LIN {X 0,Y 573.207,Z 217.084,A -85,B 0,C 180,E1 -2298.541,E2 -2298.541} C_VEL
LIN {X 0,Y 573.23,Z 217.078,A -85,B 0,C 180,E1 -2301.297,E2 -2301.297} C_VEL
LIN {X 0,Y 573.197,Z 217.089,A -85,B 0,C 180,E1 -2304.021,E2 -2304.021} C_VEL
LIN {X 0,Y 573.274,Z 217.073,A -85,B 0,C 180,E1 -2306.518,E2 -2306.518} C_VEL
LIN {X 0,Y 573.227,Z 217.085,A -85,B 0,C 180,E1 -2309.119,E2 -2309.119} C_VEL
LIN {X 0,Y 573.203,Z 217.082,A -85,B 0,C 180,E1 -2311.434,E2 -2311.434} C_VEL
LIN {X 0,Y 573.235,Z 217.079,A -85,B 0,C 180,E1 -2313.809,E2 -2313.809} C_VEL
LIN {X 0,Y 573.212,Z 217.085,A -85,B 0,C 180,E1 -2316.134,E2 -2316.134} C_VEL
LIN {X 0,Y 573.257,Z 217.076,A -85,B 0,C 180,E1 -2318.709,E2 -2318.709} C_VEL
LIN {X 0,Y 573.226,Z 217.082,A -85,B 0,C 180,E1 -2321.411,E2 -2321.411} C_VEL
LIN {X 0,Y 573.245,Z 217.077,A -85,B 0,C 180,E1 -2323.622,E2 -2323.622} C_VEL
LIN {X 0,Y 573.261,Z 217.077,A -85,B 0,C 180,E1 -2325.807,E2 -2325.807} C_VEL
LIN {X 0,Y 573.231,Z 217.078,A -85,B 0,C 180,E1 -2328.765,E2 -2328.765} C_VEL
LIN {X 0,Y 573.247,Z 217.081,A -85,B 0,C 180,E1 -2331.54,E2 -2331.54} C_VEL
LIN {X 0,Y 573.244,Z 217.077,A -85,B 0,C 180,E1 -2333.665,E2 -2333.665} C_VEL
LIN {X 0,Y 573.228,Z 217.079,A -85,B 0,C 180,E1 -2335.781,E2 -2335.781} C_VEL
LIN {X 0,Y 573.315,Z 217.072,A -85,B 0,C 180,E1 -2337.892,E2 -2337.892} C_VEL
LIN {X 0,Y 573.317,Z 217.073,A -85,B 0,C 180,E1 -2340,E2 -2340} C_VEL
LIN {X 0,Y 573.285,Z 217.072,A -85,B 0,C 180,E1 -2342.811,E2 -2342.811} C_VEL
LIN {X 0,Y 573.288,Z 217.072,A -85,B 0,C 180,E1 -2345.628,E2 -2345.628} C_VEL
LIN {X 0,Y 573.271,Z 217.074,A -85,B 0,C 180,E1 -2347.75,E2 -2347.75} C_VEL
LIN {X 0,Y 573.268,Z 217.075,A -85,B 0,C 180,E1 -2350.597,E2 -2350.597} C_VEL
LIN {X 0,Y 573.239,Z 217.077,A -85,B 0,C 180,E1 -2352.749,E2 -2352.749} C_VEL
LIN {X 0,Y 573.219,Z 217.082,A -85,B 0,C 180,E1 -2354.92,E2 -2354.92} C_VEL
LIN {X 0,Y 573.213,Z 217.08,A -85,B 0,C 180,E1 -2357.85,E2 -2357.85} C_VEL
LIN {X 0,Y 573.244,Z 217.08,A -85,B 0,C 180,E1 -2360.077,E2 -2360.077} C_VEL
LIN {X 0,Y 573.24,Z 217.081,A -85,B 0,C 180,E1 -2362.338,E2 -2362.338} C_VEL
LIN {X 0,Y 573.253,Z 217.076,A -85,B 0,C 180,E1 -2364.375,E2 -2364.375} C_VEL
LIN {X 0,Y 572.626,Z 217.155,A -85,B 0,C 180,E1 -2364.961,E2 -2364.961} C_VEL
LIN {X 0,Y 569.775,Z 217.515,A -85,B 0,C 180,E1 -2365.912,E2 -2365.912} C_VEL
LIN {X 0,Y 567.328,Z 217.822,A -85,B 0,C 180,E1 -2366.677,E2 -2366.677} C_VEL
LIN {X 0,Y 566.26,Z 217.952,A -85,B 0,C 180,E1 -2367.268,E2 -2367.268} C_VEL
LIN {X 0,Y 566.164,Z 217.962,A -85,B 0,C 180,E1 -2367.469,E2 -2367.469} C_VEL
LIN {X 0,Y 566.162,Z 217.958,A -85,B 0,C 180,E1 -2369.771,E2 -2369.771} C_VEL
LIN {X 0,Y 566.207,Z 217.959,A -85,B 0,C 180,E1 -2372.429,E2 -2372.429} C_VEL
LIN {X 0,Y 566.183,Z 217.956,A -85,B 0,C 180,E1 -2374.989,E2 -2374.989} C_VEL
LIN {X 0,Y 566.2,Z 217.96,A -85,B 0,C 180,E1 -2377.461,E2 -2377.461} C_VEL
LIN {X 0,Y 566.211,Z 217.953,A -85,B 0,C 180,E1 -2380.199,E2 -2380.199} C_VEL
LIN {X 0,Y 566.19,Z 217.957,A -85,B 0,C 180,E1 -2383.056,E2 -2383.056} C_VEL
LIN {X 0,Y 566.161,Z 217.966,A -85,B 0,C 180,E1 -2386.053,E2 -2386.053} C_VEL
LIN {X 0,Y 566.171,Z 217.958,A -85,B 0,C 180,E1 -2388.86,E2 -2388.86} C_VEL
LIN {X 0,Y 566.216,Z 217.956,A -85,B 0,C 180,E1 -2391.442,E2 -2391.442} C_VEL
LIN {X 0,Y 566.133,Z 217.966,A -85,B 0,C 180,E1 -2394.305,E2 -2394.305} C_VEL
LIN {X 0,Y 566.087,Z 217.975,A -85,B 0,C 180,E1 -2395.173,E2 -2395.173} C_VEL
LIN {X 0,Y 566.037,Z 219.577,A -85,B 0,C 180,E1 -2396.885,E2 -2396.885} C_VEL
LIN {X 0,Y 566.018,Z 222.313,A -85,B 0,C 180,E1 -2399.397,E2 -2399.397} C_VEL
LIN {X 0,Y 566,Z 224.975,A -85,B 0,C 180,E1 -2401.846,E2 -2401.846} C_VEL
LIN {X 0,Y 565.962,Z 227.66,A -85,B 0,C 180,E1 -2404.238,E2 -2404.238} C_VEL
LIN {X 0,Y 565.917,Z 230.561,A -85,B 0,C 180,E1 -2406.779,E2 -2406.779} C_VEL
LIN {X 0,Y 565.911,Z 233.852,A -85,B 0,C 180,E1 -2409.651,E2 -2409.651} C_VEL
LIN {X 0,Y 565.852,Z 237.455,A -85,B 0,C 180,E1 -2412.657,E2 -2412.657} C_VEL
LIN {X 0,Y 565.888,Z 241.317,A -85,B 0,C 180,E1 -2415.631,E2 -2415.631} C_VEL
LIN {X 0,Y 565.872,Z 243.671,A -85,B 0,C 180,E1 -2417.424,E2 -2417.424} C_VEL
LIN {X 0,Y 566.905,Z 251.271,A -85,B 0,C 180,E1 -2417.629,E2 -2417.629} C_VEL
LIN {X 0,Y 566.793,Z 263.775,A -85,B 0,C 180,E1 -2418.013,E2 -2418.013} C_VEL
LIN {X 0,Y 566.68,Z 275.32,A -85,B 0,C 180,E1 -2418.505,E2 -2418.505} C_VEL
LIN {X 0,Y 566.53,Z 287.548,A -85,B 0,C 180,E1 -2419.19,E2 -2419.19} C_VEL
LIN {X 0,Y 566.337,Z 298.841,A -85,B 0,C 180,E1 -2419.995,E2 -2419.995} C_VEL
LIN {X 0,Y 566.238,Z 308.888,A -85,B 0,C 180,E1 -2420.895,E2 -2420.895} C_VEL
LIN {X 0,Y 566.113,Z 318.589,A -85,B 0,C 180,E1 -2421.971,E2 -2421.971} C_VEL
LIN {X 0,Y 566.05,Z 325.158,A -85,B 0,C 180,E1 -2422.868,E2 -2422.868} C_VEL
LIN {X 0,Y 566.003,Z 331.626,A -85,B 0,C 180,E1 -2423.941,E2 -2423.941} C_VEL
LIN {X 0,Y 565.878,Z 336.764,A -85,B 0,C 180,E1 -2425.012,E2 -2425.012} C_VEL
LIN {X 0,Y 565.926,Z 340.753,A -85,B 0,C 180,E1 -2426.083,E2 -2426.083} C_VEL
LIN {X 0,Y 565.878,Z 343.702,A -85,B 0,C 180,E1 -2427.152,E2 -2427.152} C_VEL
LIN {X 0,Y 565.839,Z 345.127,A -85,B 0,C 180,E1 -2427.864,E2 -2427.864} C_VEL
LIN {X 0,Y 565.841,Z 346.756,A -85,B 0,C 180,E1 -2429.288,E2 -2429.288} C_VEL
LIN {X 0,Y 565.839,Z 346.996,A -85,B 0,C 180,E1 -2430,E2 -2430} C_VEL
LIN {X 0,Y 565.841,Z 346.815,A -85,B 0,C 180,E1 -2430.712,E2 -2430.712} C_VEL
LIN {X 0,Y 565.838,Z 345.268,A -85,B 0,C 180,E1 -2432.135,E2 -2432.135} C_VEL
LIN {X 0,Y 565.878,Z 343.907,A -85,B 0,C 180,E1 -2432.847,E2 -2432.847} C_VEL
LIN {X 0,Y 565.926,Z 341.03,A -85,B 0,C 180,E1 -2433.916,E2 -2433.916} C_VEL
LIN {X 0,Y 565.878,Z 337.129,A -85,B 0,C 180,E1 -2434.987,E2 -2434.987} C_VEL
LIN {X 0,Y 565.99,Z 332.097,A -85,B 0,C 180,E1 -2436.059,E2 -2436.059} C_VEL
LIN {X 0,Y 566.031,Z 325.772,A -85,B 0,C 180,E1 -2437.132,E2 -2437.132} C_VEL
LIN {X 0,Y 566.128,Z 317.85,A -85,B 0,C 180,E1 -2438.208,E2 -2438.208} C_VEL
LIN {X 0,Y 566.249,Z 307.999,A -85,B 0,C 180,E1 -2439.285,E2 -2439.285} C_VEL
LIN {X 0,Y 566.405,Z 297.68,A -85,B 0,C 180,E1 -2440.184,E2 -2440.184} C_VEL
LIN {X 0,Y 566.506,Z 286.399,A -85,B 0,C 180,E1 -2440.973,E2 -2440.973} C_VEL
LIN {X 0,Y 566.691,Z 275.188,A -85,B 0,C 180,E1 -2441.592,E2 -2441.592} C_VEL
LIN {X 0,Y 566.794,Z 262.595,A -85,B 0,C 180,E1 -2442.119,E2 -2442.119} C_VEL
LIN {X 0,Y 566.806,Z 249.418,A -85,B 0,C 180,E1 -2442.509,E2 -2442.509} C_VEL
LIN {X 0,Y 565.877,Z 243.67,A -85,B 0,C 180,E1 -2442.667,E2 -2442.667} C_VEL
LIN {X 0,Y 565.853,Z 240.455,A -85,B 0,C 180,E1 -2445.119,E2 -2445.119} C_VEL
LIN {X 0,Y 565.861,Z 237.571,A -85,B 0,C 180,E1 -2447.342,E2 -2447.342} C_VEL
LIN {X 0,Y 565.911,Z 233.953,A -85,B 0,C 180,E1 -2450.349,E2 -2450.349} C_VEL
LIN {X 0,Y 565.929,Z 230.455,A -85,B 0,C 180,E1 -2453.415,E2 -2453.415} C_VEL
LIN {X 0,Y 565.962,Z 227.765,A -85,B 0,C 180,E1 -2455.761,E2 -2455.761} C_VEL
LIN {X 0,Y 566.001,Z 225.075,A -85,B 0,C 180,E1 -2458.163,E2 -2458.163} C_VEL
LIN {X 0,Y 566.024,Z 221.935,A -85,B 0,C 180,E1 -2461.048,E2 -2461.048} C_VEL
LIN {X 0,Y 566.052,Z 218.716,A -85,B 0,C 180,E1 -2463.967,E2 -2463.967} C_VEL
LIN {X 0,Y 566.083,Z 217.975,A -85,B 0,C 180,E1 -2464.975,E2 -2464.975} C_VEL
LIN {X 0,Y 566.2,Z 217.958,A -85,B 0,C 180,E1 -2467.461,E2 -2467.461} C_VEL
LIN {X 0,Y 566.211,Z 217.955,A -85,B 0,C 180,E1 -2470.199,E2 -2470.199} C_VEL
LIN {X 0,Y 566.19,Z 217.955,A -85,B 0,C 180,E1 -2473.056,E2 -2473.056} C_VEL
LIN {X 0,Y 566.16,Z 217.962,A -85,B 0,C 180,E1 -2476.053,E2 -2476.053} C_VEL
LIN {X 0,Y 566.169,Z 217.961,A -85,B 0,C 180,E1 -2478.86,E2 -2478.86} C_VEL
LIN {X 0,Y 566.212,Z 217.954,A -85,B 0,C 180,E1 -2481.442,E2 -2481.442} C_VEL
LIN {X 0,Y 566.166,Z 217.964,A -85,B 0,C 180,E1 -2484.308,E2 -2484.308} C_VEL
LIN {X 0,Y 566.206,Z 217.953,A -85,B 0,C 180,E1 -2486.897,E2 -2486.897} C_VEL
LIN {X 0,Y 566.163,Z 217.965,A -85,B 0,C 180,E1 -2489.406,E2 -2489.406} C_VEL
LIN {X 0,Y 566.173,Z 217.958,A -85,B 0,C 180,E1 -2491.855,E2 -2491.855} C_VEL
LIN {X 0,Y 566.212,Z 217.956,A -85,B 0,C 180,E1 -2494.251,E2 -2494.251} C_VEL
LIN {X 0,Y 566.176,Z 217.959,A -85,B 0,C 180,E1 -2496.718,E2 -2496.718} C_VEL
LIN {X 0,Y 566.21,Z 217.959,A -85,B 0,C 180,E1 -2499.663,E2 -2499.663} C_VEL
LIN {X 0,Y 566.178,Z 217.957,A -85,B 0,C 180,E1 -2501.921,E2 -2501.921} C_VEL
LIN {X 0,Y 566.185,Z 217.962,A -85,B 0,C 180,E1 -2504.89,E2 -2504.89} C_VEL
LIN {X 0,Y 566.238,Z 217.952,A -85,B 0,C 180,E1 -2507.819,E2 -2507.819} C_VEL
LIN {X 0,Y 566.212,Z 217.953,A -85,B 0,C 180,E1 -2510.714,E2 -2510.714} C_VEL
LIN {X 0,Y 566.264,Z 217.951,A -85,B 0,C 180,E1 -2513.168,E2 -2513.168} C_VEL
LIN {X 0,Y 566.157,Z 217.959,A -85,B 0,C 180,E1 -2515.729,E2 -2515.729} C_VEL
LIN {X 0,Y 566.26,Z 217.946,A -85,B 0,C 180,E1 -2517.866,E2 -2517.866} C_VEL
LIN {X 0,Y 566.3,Z 217.943,A -85,B 0,C 180,E1 -2520.711,E2 -2520.711} C_VEL
LIN {X 0,Y 566.273,Z 217.945,A -85,B 0,C 180,E1 -2522.846,E2 -2522.846} C_VEL
LIN {X 0,Y 566.261,Z 217.949,A -85,B 0,C 180,E1 -2525.698,E2 -2525.698} C_VEL
LIN {X 0,Y 566.2,Z 217.96,A -85,B 0,C 180,E1 -2528.566,E2 -2528.566} C_VEL
LIN {X 0,Y 566.195,Z 217.954,A -85,B 0,C 180,E1 -2531.455,E2 -2531.455} C_VEL
LIN {X 0,Y 566.225,Z 217.951,A -85,B 0,C 180,E1 -2534.501,E2 -2534.501} C_VEL
LIN {X 0,Y 566.204,Z 217.96,A -85,B 0,C 180,E1 -2537.332,E2 -2537.332} C_VEL
LIN {X 0,Y 566.212,Z 217.956,A -85,B 0,C 180,E1 -2540.337,E2 -2540.337} C_VEL
LIN {X 0,Y 566.168,Z 217.958,A -85,B 0,C 180,E1 -2543.28,E2 -2543.28} C_VEL
LIN {X 0,Y 566.181,Z 217.963,A -85,B 0,C 180,E1 -2545.751,E2 -2545.751} C_VEL
LIN {X 0,Y 566.152,Z 217.96,A -85,B 0,C 180,E1 -2548.192,E2 -2548.192} C_VEL
LIN {X 0,Y 566.192,Z 217.961,A -85,B 0,C 180,E1 -2551.076,E2 -2551.076} C_VEL
LIN {X 0,Y 566.215,Z 217.953,A -85,B 0,C 180,E1 -2553.734,E2 -2553.734} C_VEL
LIN {X 0,Y 566.184,Z 217.957,A -85,B 0,C 180,E1 -2556.571,E2 -2556.571} C_VEL
LIN {X 0,Y 566.206,Z 217.957,A -85,B 0,C 180,E1 -2559.684,E2 -2559.684} C_VEL
LIN {X 0,Y 566.196,Z 217.96,A -85,B 0,C 180,E1 -2563.055,E2 -2563.055} C_VEL
LIN {X 0,Y 566.196,Z 217.959,A -85,B 0,C 180,E1 -2566.049,E2 -2566.049} C_VEL
LIN {X 0,Y 566.206,Z 217.956,A -85,B 0,C 180,E1 -2569.215,E2 -2569.215} C_VEL
LIN {X 0,Y 566.181,Z 217.963,A -85,B 0,C 180,E1 -2571.636,E2 -2571.636} C_VEL
LIN {X 0,Y 566.222,Z 218.101,A -85,B 0,C 180,E1 -2573.043,E2 -2573.043} C_VEL
LIN {X 0,Y 566.785,Z 221.916,A -85,B 0,C 180,E1 -2574.353,E2 -2574.353} C_VEL
LIN {X 0,Y 566.802,Z 228.679,A -85,B 0,C 180,E1 -2576.557,E2 -2576.557} C_VEL
LIN {X 0,Y 566.628,Z 237.803,A -85,B 0,C 180,E1 -2579.434,E2 -2579.434} C_VEL
LIN {X 0,Y 566.521,Z 248.394,A -85,B 0,C 180,E1 -2582.677,E2 -2582.677} C_VEL
LIN {X 0,Y 566.391,Z 257.662,A -85,B 0,C 180,E1 -2585.438,E2 -2585.438} C_VEL
LIN {X 0,Y 566.323,Z 266.929,A -85,B 0,C 180,E1 -2588.143,E2 -2588.143} C_VEL
LIN {X 0,Y 566.185,Z 277.52,A -85,B 0,C 180,E1 -2591.172,E2 -2591.172} C_VEL
LIN {X 0,Y 566.109,Z 288.112,A -85,B 0,C 180,E1 -2594.15,E2 -2594.15} C_VEL
LIN {X 0,Y 565.996,Z 299.365,A -85,B 0,C 180,E1 -2597.267,E2 -2597.267} C_VEL
LIN {X 0,Y 565.987,Z 299.53,A -85,B 0,C 180,E1 -2597.313,E2 -2597.313} C_VEL
LIN {X 0,Y 566.928,Z 306.372,A -85,B 0,C 180,E1 -2597.471,E2 -2597.471} C_VEL
LIN {X 0,Y 566.837,Z 318.498,A -85,B 0,C 180,E1 -2597.787,E2 -2597.787} C_VEL
LIN {X 0,Y 566.679,Z 330.32,A -85,B 0,C 180,E1 -2598.228,E2 -2598.228} C_VEL
LIN {X 0,Y 566.549,Z 341.713,A -85,B 0,C 180,E1 -2598.795,E2 -2598.795} C_VEL
LIN {X 0,Y 566.421,Z 353.479,A -85,B 0,C 180,E1 -2599.545,E2 -2599.545} C_VEL
LIN {X 0,Y 566.3,Z 363.647,A -85,B 0,C 180,E1 -2600.355,E2 -2600.355} C_VEL
LIN {X 0,Y 566.166,Z 372.787,A -85,B 0,C 180,E1 -2601.254,E2 -2601.254} C_VEL
LIN {X 0,Y 566.08,Z 381.691,A -85,B 0,C 180,E1 -2602.33,E2 -2602.33} C_VEL
LIN {X 0,Y 565.967,Z 388.956,A -85,B 0,C 180,E1 -2603.422,E2 -2603.422} C_VEL
LIN {X 0,Y 566.004,Z 393.681,A -85,B 0,C 180,E1 -2604.299,E2 -2604.299} C_VEL
LIN {X 0,Y 565.933,Z 398.372,A -85,B 0,C 180,E1 -2605.37,E2 -2605.37} C_VEL
LIN {X 0,Y 565.927,Z 401.957,A -85,B 0,C 180,E1 -2606.44,E2 -2606.44} C_VEL
LIN {X 0,Y 565.878,Z 403.809,A -85,B 0,C 180,E1 -2607.153,E2 -2607.153} C_VEL
LIN {X 0,Y 565.841,Z 405.2,A -85,B 0,C 180,E1 -2607.865,E2 -2607.865} C_VEL
LIN {X 0,Y 565.841,Z 406.784,A -85,B 0,C 180,E1 -2609.288,E2 -2609.288} C_VEL
LIN {X 0,Y 565.839,Z 407,A -85,B 0,C 180,E1 -2610,E2 -2610} C_VEL
LIN {X 0,Y 565.846,Z 406.185,A -85,B 0,C 180,E1 -2611.424,E2 -2611.424} C_VEL
LIN {X 0,Y 565.841,Z 405.201,A -85,B 0,C 180,E1 -2612.136,E2 -2612.136} C_VEL
LIN {X 0,Y 565.878,Z 403.809,A -85,B 0,C 180,E1 -2612.848,E2 -2612.848} C_VEL
LIN {X 0,Y 565.926,Z 400.896,A -85,B 0,C 180,E1 -2613.917,E2 -2613.917} C_VEL
LIN {X 0,Y 565.878,Z 396.949,A -85,B 0,C 180,E1 -2614.988,E2 -2614.988} C_VEL
LIN {X 0,Y 566.002,Z 391.866,A -85,B 0,C 180,E1 -2616.059,E2 -2616.059} C_VEL
LIN {X 0,Y 566.04,Z 385.469,A -85,B 0,C 180,E1 -2617.132,E2 -2617.132} C_VEL
LIN {X 0,Y 566.134,Z 377.477,A -85,B 0,C 180,E1 -2618.208,E2 -2618.208} C_VEL
LIN {X 0,Y 566.229,Z 369.335,A -85,B 0,C 180,E1 -2619.106,E2 -2619.106} C_VEL
LIN {X 0,Y 566.336,Z 359.4,A -85,B 0,C 180,E1 -2620.005,E2 -2620.005} C_VEL
LIN {X 0,Y 566.471,Z 348.326,A -85,B 0,C 180,E1 -2620.806,E2 -2620.806} C_VEL
LIN {X 0,Y 566.609,Z 335.947,A -85,B 0,C 180,E1 -2621.51,E2 -2621.51} C_VEL
LIN {X 0,Y 566.779,Z 323.762,A -85,B 0,C 180,E1 -2622.033,E2 -2622.033} C_VEL
LIN {X 0,Y 566.924,Z 310.342,A -85,B 0,C 180,E1 -2622.439,E2 -2622.439} C_VEL
LIN {X 0,Y 566.636,Z 303.508,A -85,B 0,C 180,E1 -2622.593,E2 -2622.593} C_VEL
LIN {X 0,Y 565.987,Z 299.53,A -85,B 0,C 180,E1 -2622.687,E2 -2622.687} C_VEL
LIN {X 0,Y 566.085,Z 289.435,A -85,B 0,C 180,E1 -2625.482,E2 -2625.482} C_VEL
LIN {X 0,Y 566.159,Z 278.843,A -85,B 0,C 180,E1 -2628.454,E2 -2628.454} C_VEL
LIN {X 0,Y 566.246,Z 269.576,A -85,B 0,C 180,E1 -2631.096,E2 -2631.096} C_VEL
LIN {X 0,Y 566.365,Z 260.309,A -85,B 0,C 180,E1 -2633.784,E2 -2633.784} C_VEL
LIN {X 0,Y 566.488,Z 251.041,A -85,B 0,C 180,E1 -2636.528,E2 -2636.528} C_VEL
LIN {X 0,Y 566.569,Z 241.774,A -85,B 0,C 180,E1 -2639.339,E2 -2639.339} C_VEL
LIN {X 0,Y 566.75,Z 232.507,A -85,B 0,C 180,E1 -2642.224,E2 -2642.224} C_VEL
LIN {X 0,Y 566.839,Z 223.615,A -85,B 0,C 180,E1 -2645.084,E2 -2645.084} C_VEL
LIN {X 0,Y 566.305,Z 218.597,A -85,B 0,C 180,E1 -2646.784,E2 -2646.784} C_VEL
LIN {X 0,Y 566.183,Z 217.963,A -85,B 0,C 180,E1 -2647.016,E2 -2647.016} C_VEL
LIN {X 0,Y 566.215,Z 217.955,A -85,B 0,C 180,E1 -2649.685,E2 -2649.685} C_VEL
LIN {X 0,Y 566.205,Z 217.955,A -85,B 0,C 180,E1 -2652.917,E2 -2652.917} C_VEL
LIN {X 0,Y 566.197,Z 217.955,A -85,B 0,C 180,E1 -2656.05,E2 -2656.05} C_VEL
LIN {X 0,Y 566.155,Z 217.966,A -85,B 0,C 180,E1 -2658.858,E2 -2658.858} C_VEL
LIN {X 0,Y 566.201,Z 217.954,A -85,B 0,C 180,E1 -2661.444,E2 -2661.444} C_VEL
LIN {X 0,Y 566.154,Z 217.963,A -85,B 0,C 180,E1 -2664.307,E2 -2664.307} C_VEL
LIN {X 0,Y 566.225,Z 217.953,A -85,B 0,C 180,E1 -2666.898,E2 -2666.898} C_VEL
LIN {X 0,Y 566.175,Z 217.96,A -85,B 0,C 180,E1 -2669.407,E2 -2669.407} C_VEL
LIN {X 0,Y 566.155,Z 217.96,A -85,B 0,C 180,E1 -2671.854,E2 -2671.854} C_VEL
LIN {X 0,Y 566.182,Z 217.963,A -85,B 0,C 180,E1 -2674.249,E2 -2674.249} C_VEL
LIN {X 0,Y 566.181,Z 217.96,A -85,B 0,C 180,E1 -2677.368,E2 -2677.368} C_VEL
LIN {X 0,Y 566.213,Z 217.956,A -85,B 0,C 180,E1 -2679.663,E2 -2679.663} C_VEL
LIN {X 0,Y 566.205,Z 217.96,A -85,B 0,C 180,E1 -2682.668,E2 -2682.668} C_VEL
LIN {X 0,Y 566.225,Z 217.952,A -85,B 0,C 180,E1 -2685.627,E2 -2685.627} C_VEL
LIN {X 0,Y 566.193,Z 217.954,A -85,B 0,C 180,E1 -2688.7,E2 -2688.7} C_VEL
LIN {X 0,Y 566.2,Z 217.96,A -85,B 0,C 180,E1 -2691.434,E2 -2691.434} C_VEL
LIN {X 0,Y 566.261,Z 217.949,A -85,B 0,C 180,E1 -2694.302,E2 -2694.302} C_VEL
LIN {X 0,Y 566.286,Z 217.947,A -85,B 0,C 180,E1 -2697.866,E2 -2697.866} C_VEL
LIN {X 0,Y 566.286,Z 217.948,A -85,B 0,C 180,E1 -2700,E2 -2700} C_VEL
LIN {X 0,Y 566.254,Z 217.948,A -85,B 0,C 180,E1 -2702.846,E2 -2702.846} C_VEL
LIN {X 0,Y 566.255,Z 217.947,A -85,B 0,C 180,E1 -2705.698,E2 -2705.698} C_VEL
LIN {X 0,Y 566.206,Z 217.959,A -85,B 0,C 180,E1 -2708.566,E2 -2708.566} C_VEL
LIN {X 0,Y 566.248,Z 217.951,A -85,B 0,C 180,E1 -2711.454,E2 -2711.454} C_VEL
LIN {X 0,Y 566.21,Z 217.953,A -85,B 0,C 180,E1 -2714.494,E2 -2714.494} C_VEL
LIN {X 0,Y 566.176,Z 217.959,A -85,B 0,C 180,E1 -2717.332,E2 -2717.332} C_VEL
LIN {X 0,Y 566.207,Z 217.953,A -85,B 0,C 180,E1 -2719.581,E2 -2719.581} C_VEL
LIN {X 0,Y 566.199,Z 217.958,A -85,B 0,C 180,E1 -2721.862,E2 -2721.862} C_VEL
LIN {X 0,Y 566.224,Z 217.953,A -85,B 0,C 180,E1 -2725.03,E2 -2725.03} C_VEL
LIN {X 0,Y 566.164,Z 217.962,A -85,B 0,C 180,E1 -2727.469,E2 -2727.469} C_VEL
LIN {X 0,Y 565.471,Z 218.046,A -85,B 0,C 180,E1 -2728.063,E2 -2728.063} C_VEL
LIN {X 0,Y 562.595,Z 218.408,A -85,B 0,C 180,E1 -2729.026,E2 -2729.026} C_VEL
LIN {X 0,Y 560.194,Z 218.705,A -85,B 0,C 180,E1 -2729.802,E2 -2729.802} C_VEL
LIN {X 0,Y 559.184,Z 218.832,A -85,B 0,C 180,E1 -2730.401,E2 -2730.401} C_VEL
LIN {X 0,Y 559.112,Z 218.837,A -85,B 0,C 180,E1 -2730.603,E2 -2730.603} C_VEL
LIN {X 0,Y 559.157,Z 218.834,A -85,B 0,C 180,E1 -2732.715,E2 -2732.715} C_VEL
LIN {X 0,Y 559.132,Z 218.836,A -85,B 0,C 180,E1 -2735.324,E2 -2735.324} C_VEL
LIN {X 0,Y 559.136,Z 218.836,A -85,B 0,C 180,E1 -2738.018,E2 -2738.018} C_VEL
LIN {X 0,Y 559.158,Z 218.838,A -85,B 0,C 180,E1 -2740.813,E2 -2740.813} C_VEL
LIN {X 0,Y 559.113,Z 218.838,A -85,B 0,C 180,E1 -2743.737,E2 -2743.737} C_VEL
LIN {X 0,Y 559.112,Z 218.841,A -85,B 0,C 180,E1 -2746.263,E2 -2746.263} C_VEL
LIN {X 0,Y 559.157,Z 218.835,A -85,B 0,C 180,E1 -2749.187,E2 -2749.187} C_VEL
LIN {X 0,Y 559.137,Z 218.834,A -85,B 0,C 180,E1 -2751.982,E2 -2751.982} C_VEL
LIN {X 0,Y 559.063,Z 218.849,A -85,B 0,C 180,E1 -2754.671,E2 -2754.671} C_VEL
LIN {X 0,Y 558.991,Z 218.859,A -85,B 0,C 180,E1 -2755.544,E2 -2755.544} C_VEL
LIN {X 0,Y 558.949,Z 221.603,A -85,B 0,C 180,E1 -2758.123,E2 -2758.123} C_VEL
LIN {X 0,Y 558.92,Z 224.314,A -85,B 0,C 180,E1 -2760.633,E2 -2760.633} C_VEL
LIN {X 0,Y 558.913,Z 227.149,A -85,B 0,C 180,E1 -2763.226,E2 -2763.226} C_VEL
LIN {X 0,Y 558.86,Z 229.66,A -85,B 0,C 180,E1 -2765.481,E2 -2765.481} C_VEL
LIN {X 0,Y 558.838,Z 233.164,A -85,B 0,C 180,E1 -2768.534,E2 -2768.534} C_VEL
LIN {X 0,Y 558.796,Z 235.9,A -85,B 0,C 180,E1 -2770.913,E2 -2770.913} C_VEL
LIN {X 0,Y 558.764,Z 239.378,A -85,B 0,C 180,E1 -2773.936,E2 -2773.936} C_VEL
LIN {X 0,Y 558.777,Z 242.26,A -85,B 0,C 180,E1 -2776.174,E2 -2776.174} C_VEL
LIN {X 0,Y 558.783,Z 243.672,A -85,B 0,C 180,E1 -2777.262,E2 -2777.262} C_VEL
LIN {X 0,Y 559.971,Z 252.207,A -85,B 0,C 180,E1 -2777.496,E2 -2777.496} C_VEL
LIN {X 0,Y 559.854,Z 264.292,A -85,B 0,C 180,E1 -2777.88,E2 -2777.88} C_VEL
LIN {X 0,Y 559.688,Z 276.303,A -85,B 0,C 180,E1 -2778.41,E2 -2778.41} C_VEL
LIN {X 0,Y 559.54,Z 287.647,A -85,B 0,C 180,E1 -2779.06,E2 -2779.06} C_VEL
LIN {X 0,Y 559.349,Z 298.849,A -85,B 0,C 180,E1 -2779.869,E2 -2779.869} C_VEL
LIN {X 0,Y 559.211,Z 308.893,A -85,B 0,C 180,E1 -2780.779,E2 -2780.779} C_VEL
LIN {X 0,Y 559.051,Z 318.594,A -85,B 0,C 180,E1 -2781.869,E2 -2781.869} C_VEL
LIN {X 0,Y 558.971,Z 326.455,A -85,B 0,C 180,E1 -2782.977,E2 -2782.977} C_VEL
LIN {X 0,Y 558.936,Z 333.453,A -85,B 0,C 180,E1 -2784.227,E2 -2784.227} C_VEL
LIN {X 0,Y 558.826,Z 338.194,A -85,B 0,C 180,E1 -2785.311,E2 -2785.311} C_VEL
LIN {X 0,Y 558.836,Z 341.828,A -85,B 0,C 180,E1 -2786.395,E2 -2786.395} C_VEL
LIN {X 0,Y 558.799,Z 343.704,A -85,B 0,C 180,E1 -2787.116,E2 -2787.116} C_VEL
LIN {X 0,Y 558.745,Z 345.127,A -85,B 0,C 180,E1 -2787.837,E2 -2787.837} C_VEL
LIN {X 0,Y 558.741,Z 346.757,A -85,B 0,C 180,E1 -2789.279,E2 -2789.279} C_VEL
LIN {X 0,Y 558.74,Z 346.996,A -85,B 0,C 180,E1 -2790,E2 -2790} C_VEL
LIN {X 0,Y 558.741,Z 346.815,A -85,B 0,C 180,E1 -2790.721,E2 -2790.721} C_VEL
LIN {X 0,Y 558.745,Z 345.266,A -85,B 0,C 180,E1 -2792.162,E2 -2792.162} C_VEL
LIN {X 0,Y 558.8,Z 343.905,A -85,B 0,C 180,E1 -2792.884,E2 -2792.884} C_VEL
LIN {X 0,Y 558.844,Z 341.028,A -85,B 0,C 180,E1 -2793.966,E2 -2793.966} C_VEL
LIN {X 0,Y 558.798,Z 337.127,A -85,B 0,C 180,E1 -2795.051,E2 -2795.051} C_VEL
LIN {X 0,Y 558.91,Z 332.094,A -85,B 0,C 180,E1 -2796.136,E2 -2796.136} C_VEL
LIN {X 0,Y 558.972,Z 325.768,A -85,B 0,C 180,E1 -2797.223,E2 -2797.223} C_VEL
LIN {X 0,Y 559.091,Z 317.845,A -85,B 0,C 180,E1 -2798.312,E2 -2798.312} C_VEL
LIN {X 0,Y 559.223,Z 307.992,A -85,B 0,C 180,E1 -2799.403,E2 -2799.403} C_VEL
LIN {X 0,Y 559.399,Z 297.672,A -85,B 0,C 180,E1 -2800.313,E2 -2800.313} C_VEL
LIN {X 0,Y 559.529,Z 286.641,A -85,B 0,C 180,E1 -2801.095,E2 -2801.095} C_VEL
LIN {X 0,Y 559.712,Z 276.453,A -85,B 0,C 180,E1 -2801.672,E2 -2801.672} C_VEL
LIN {X 0,Y 559.818,Z 264.962,A -85,B 0,C 180,E1 -2802.185,E2 -2802.185} C_VEL
LIN {X 0,Y 559.986,Z 252.141,A -85,B 0,C 180,E1 -2802.595,E2 -2802.595} C_VEL
LIN {X 0,Y 558.767,Z 243.669,A -85,B 0,C 180,E1 -2802.831,E2 -2802.831} C_VEL
LIN {X 0,Y 558.751,Z 240.454,A -85,B 0,C 180,E1 -2805.316,E2 -2805.316} C_VEL
LIN {X 0,Y 558.772,Z 237.741,A -85,B 0,C 180,E1 -2807.569,E2 -2807.569} C_VEL
LIN {X 0,Y 558.817,Z 235.133,A -85,B 0,C 180,E1 -2809.851,E2 -2809.851} C_VEL
LIN {X 0,Y 558.809,Z 232.439,A -85,B 0,C 180,E1 -2812.167,E2 -2812.167} C_VEL
LIN {X 0,Y 558.882,Z 229.101,A -85,B 0,C 180,E1 -2815.121,E2 -2815.121} C_VEL
LIN {X 0,Y 558.906,Z 226.202,A -85,B 0,C 180,E1 -2817.727,E2 -2817.727} C_VEL
LIN {X 0,Y 558.96,Z 223.52,A -85,B 0,C 180,E1 -2820.194,E2 -2820.194} C_VEL
LIN {X 0,Y 558.964,Z 220.788,A -85,B 0,C 180,E1 -2822.728,E2 -2822.728} C_VEL
LIN {X 0,Y 558.988,Z 218.861,A -85,B 0,C 180,E1 -2824.456,E2 -2824.456} C_VEL
LIN {X 0,Y 559.141,Z 218.839,A -85,B 0,C 180,E1 -2827.109,E2 -2827.109} C_VEL
LIN {X 0,Y 559.165,Z 218.831,A -85,B 0,C 180,E1 -2829.942,E2 -2829.942} C_VEL
LIN {X 0,Y 559.153,Z 218.833,A -85,B 0,C 180,E1 -2832.744,E2 -2832.744} C_VEL
LIN {X 0,Y 559.126,Z 218.842,A -85,B 0,C 180,E1 -2835.764,E2 -2835.764} C_VEL
LIN {X 0,Y 559.157,Z 218.832,A -85,B 0,C 180,E1 -2838.229,E2 -2838.229} C_VEL
LIN {X 0,Y 559.176,Z 218.833,A -85,B 0,C 180,E1 -2841.192,E2 -2841.192} C_VEL
LIN {X 0,Y 559.143,Z 218.835,A -85,B 0,C 180,E1 -2843.789,E2 -2843.789} C_VEL
LIN {X 0,Y 559.151,Z 218.834,A -85,B 0,C 180,E1 -2846.424,E2 -2846.424} C_VEL
LIN {X 0,Y 559.147,Z 218.834,A -85,B 0,C 180,E1 -2848.98,E2 -2848.98} C_VEL
LIN {X 0,Y 559.115,Z 218.838,A -85,B 0,C 180,E1 -2851.63,E2 -2851.63} C_VEL
LIN {X 0,Y 559.177,Z 218.83,A -85,B 0,C 180,E1 -2853.903,E2 -2853.903} C_VEL
LIN {X 0,Y 559.145,Z 218.836,A -85,B 0,C 180,E1 -2856.571,E2 -2856.571} C_VEL
LIN {X 0,Y 559.18,Z 218.832,A -85,B 0,C 180,E1 -2859.395,E2 -2859.395} C_VEL
LIN {X 0,Y 559.129,Z 218.837,A -85,B 0,C 180,E1 -2861.685,E2 -2861.685} C_VEL
LIN {X 0,Y 559.14,Z 218.833,A -85,B 0,C 180,E1 -2863.947,E2 -2863.947} C_VEL
LIN {X 0,Y 559.153,Z 218.834,A -85,B 0,C 180,E1 -2866.924,E2 -2866.924} C_VEL
LIN {X 0,Y 559.197,Z 218.827,A -85,B 0,C 180,E1 -2869.133,E2 -2869.133} C_VEL
LIN {X 0,Y 559.199,Z 218.828,A -85,B 0,C 180,E1 -2872.053,E2 -2872.053} C_VEL
LIN {X 0,Y 559.246,Z 218.827,A -85,B 0,C 180,E1 -2874.953,E2 -2874.953} C_VEL
LIN {X 0,Y 559.234,Z 218.822,A -85,B 0,C 180,E1 -2877.839,E2 -2877.839} C_VEL
LIN {X 0,Y 559.27,Z 218.818,A -85,B 0,C 180,E1 -2880.72,E2 -2880.72} C_VEL
LIN {X 0,Y 559.239,Z 218.822,A -85,B 0,C 180,E1 -2882.881,E2 -2882.881} C_VEL
LIN {X 0,Y 559.23,Z 218.824,A -85,B 0,C 180,E1 -2885.77,E2 -2885.77} C_VEL
LIN {X 0,Y 559.165,Z 218.837,A -85,B 0,C 180,E1 -2888.675,E2 -2888.675} C_VEL
LIN {X 0,Y 559.157,Z 218.832,A -85,B 0,C 180,E1 -2891.601,E2 -2891.601} C_VEL
LIN {X 0,Y 559.184,Z 218.828,A -85,B 0,C 180,E1 -2894.588,E2 -2894.588} C_VEL
LIN {X 0,Y 559.163,Z 218.834,A -85,B 0,C 180,E1 -2897.557,E2 -2897.557} C_VEL
LIN {X 0,Y 559.17,Z 218.83,A -85,B 0,C 180,E1 -2899.838,E2 -2899.838} C_VEL
LIN {X 0,Y 559.143,Z 218.838,A -85,B 0,C 180,E1 -2902.153,E2 -2902.153} C_VEL
LIN {X 0,Y 559.14,Z 218.834,A -85,B 0,C 180,E1 -2905.178,E2 -2905.178} C_VEL
LIN {X 0,Y 559.109,Z 218.842,A -85,B 0,C 180,E1 -2907.716,E2 -2907.716} C_VEL
LIN {X 0,Y 559.141,Z 218.834,A -85,B 0,C 180,E1 -2910.184,E2 -2910.184} C_VEL
LIN {X 0,Y 559.161,Z 218.837,A -85,B 0,C 180,E1 -2912.715,E2 -2912.715} C_VEL
LIN {X 0,Y 559.126,Z 218.836,A -85,B 0,C 180,E1 -2915.324,E2 -2915.324} C_VEL
LIN {X 0,Y 559.128,Z 218.839,A -85,B 0,C 180,E1 -2918.018,E2 -2918.018} C_VEL
LIN {X 0,Y 559.117,Z 218.838,A -85,B 0,C 180,E1 -2920.816,E2 -2920.816} C_VEL
LIN {X 0,Y 559.138,Z 218.834,A -85,B 0,C 180,E1 -2923.734,E2 -2923.734} C_VEL
LIN {X 0,Y 559.148,Z 218.835,A -85,B 0,C 180,E1 -2926.804,E2 -2926.804} C_VEL
LIN {X 0,Y 559.158,Z 218.834,A -85,B 0,C 180,E1 -2929.188,E2 -2929.188} C_VEL
LIN {X 0,Y 559.13,Z 218.84,A -85,B 0,C 180,E1 -2931.982,E2 -2931.982} C_VEL
LIN {X 0,Y 559.18,Z 218.95,A -85,B 0,C 180,E1 -2932.797,E2 -2932.797} C_VEL
LIN {X 0,Y 559.838,Z 223.235,A -85,B 0,C 180,E1 -2934.286,E2 -2934.286} C_VEL
LIN {X 0,Y 559.848,Z 229.86,A -85,B 0,C 180,E1 -2936.471,E2 -2936.471} C_VEL
LIN {X 0,Y 559.679,Z 237.803,A -85,B 0,C 180,E1 -2939.013,E2 -2939.013} C_VEL
LIN {X 0,Y 559.557,Z 247.155,A -85,B 0,C 180,E1 -2941.927,E2 -2941.927} C_VEL
LIN {X 0,Y 559.406,Z 256.509,A -85,B 0,C 180,E1 -2944.765,E2 -2944.765} C_VEL
LIN {X 0,Y 559.291,Z 265.605,A -85,B 0,C 180,E1 -2947.464,E2 -2947.464} C_VEL
LIN {X 0,Y 559.179,Z 276.036,A -85,B 0,C 180,E1 -2950.499,E2 -2950.499} C_VEL
LIN {X 0,Y 559.052,Z 286.788,A -85,B 0,C 180,E1 -2953.569,E2 -2953.569} C_VEL
LIN {X 0,Y 558.954,Z 297.379,A -85,B 0,C 180,E1 -2956.549,E2 -2956.549} C_VEL
LIN {X 0,Y 558.933,Z 299.53,A -85,B 0,C 180,E1 -2957.15,E2 -2957.15} C_VEL
LIN {X 0,Y 560.012,Z 307.511,A -85,B 0,C 180,E1 -2957.336,E2 -2957.336} C_VEL
LIN {X 0,Y 559.896,Z 319.878,A -85,B 0,C 180,E1 -2957.679,E2 -2957.679} C_VEL
LIN {X 0,Y 559.718,Z 332.283,A -85,B 0,C 180,E1 -2958.171,E2 -2958.171} C_VEL
LIN {X 0,Y 559.541,Z 343.912,A -85,B 0,C 180,E1 -2958.782,E2 -2958.782} C_VEL
LIN {X 0,Y 559.433,Z 354.747,A -85,B 0,C 180,E1 -2959.504,E2 -2959.504} C_VEL
LIN {X 0,Y 559.243,Z 365.601,A -85,B 0,C 180,E1 -2960.415,E2 -2960.415} C_VEL
LIN {X 0,Y 559.127,Z 374.414,A -85,B 0,C 180,E1 -2961.325,E2 -2961.325} C_VEL
LIN {X 0,Y 558.996,Z 383.001,A -85,B 0,C 180,E1 -2962.414,E2 -2962.414} C_VEL
LIN {X 0,Y 558.885,Z 390.688,A -85,B 0,C 180,E1 -2963.649,E2 -2963.649} C_VEL
LIN {X 0,Y 558.869,Z 395.366,A -85,B 0,C 180,E1 -2964.588,E2 -2964.588} C_VEL
LIN {X 0,Y 558.868,Z 399.678,A -85,B 0,C 180,E1 -2965.673,E2 -2965.673} C_VEL
LIN {X 0,Y 558.836,Z 401.957,A -85,B 0,C 180,E1 -2966.395,E2 -2966.395} C_VEL
LIN {X 0,Y 558.799,Z 403.809,A -85,B 0,C 180,E1 -2967.116,E2 -2967.116} C_VEL
LIN {X 0,Y 558.746,Z 405.2,A -85,B 0,C 180,E1 -2967.838,E2 -2967.838} C_VEL
LIN {X 0,Y 558.741,Z 406.785,A -85,B 0,C 180,E1 -2969.279,E2 -2969.279} C_VEL
LIN {X 0,Y 558.74,Z 407,A -85,B 0,C 180,E1 -2970,E2 -2970} C_VEL
LIN {X 0,Y 558.745,Z 406.185,A -85,B 0,C 180,E1 -2971.442,E2 -2971.442} C_VEL
LIN {X 0,Y 558.746,Z 405.2,A -85,B 0,C 180,E1 -2972.163,E2 -2972.163} C_VEL
LIN {X 0,Y 558.799,Z 403.809,A -85,B 0,C 180,E1 -2972.884,E2 -2972.884} C_VEL
LIN {X 0,Y 558.844,Z 400.896,A -85,B 0,C 180,E1 -2973.966,E2 -2973.966} C_VEL
LIN {X 0,Y 558.798,Z 396.949,A -85,B 0,C 180,E1 -2975.051,E2 -2975.051} C_VEL
LIN {X 0,Y 558.922,Z 391.866,A -85,B 0,C 180,E1 -2976.136,E2 -2976.136} C_VEL
LIN {X 0,Y 558.977,Z 385.468,A -85,B 0,C 180,E1 -2977.223,E2 -2977.223} C_VEL
LIN {X 0,Y 559.099,Z 377.477,A -85,B 0,C 180,E1 -2978.312,E2 -2978.312} C_VEL
LIN {X 0,Y 559.195,Z 369.335,A -85,B 0,C 180,E1 -2979.221,E2 -2979.221} C_VEL
LIN {X 0,Y 559.335,Z 359.4,A -85,B 0,C 180,E1 -2980.132,E2 -2980.132} C_VEL
LIN {X 0,Y 559.476,Z 348.435,A -85,B 0,C 180,E1 -2980.936,E2 -2980.936} C_VEL
LIN {X 0,Y 559.636,Z 336.819,A -85,B 0,C 180,E1 -2981.61,E2 -2981.61} C_VEL
LIN {X 0,Y 559.81,Z 324.983,A -85,B 0,C 180,E1 -2982.139,E2 -2982.139} C_VEL
LIN {X 0,Y 559.998,Z 312.17,A -85,B 0,C 180,E1 -2982.549,E2 -2982.549} C_VEL
LIN {X 0,Y 559.808,Z 304.935,A -85,B 0,C 180,E1 -2982.72,E2 -2982.72} C_VEL
LIN {X 0,Y 558.933,Z 299.53,A -85,B 0,C 180,E1 -2982.85,E2 -2982.85} C_VEL
LIN {X 0,Y 559.05,Z 289.435,A -85,B 0,C 180,E1 -2985.681,E2 -2985.681} C_VEL
LIN {X 0,Y 559.129,Z 278.843,A -85,B 0,C 180,E1 -2988.695,E2 -2988.695} C_VEL
LIN {X 0,Y 559.227,Z 268.915,A -85,B 0,C 180,E1 -2991.567,E2 -2991.567} C_VEL
LIN {X 0,Y 559.387,Z 258.985,A -85,B 0,C 180,E1 -2994.495,E2 -2994.495} C_VEL
LIN {X 0,Y 559.519,Z 249.719,A -85,B 0,C 180,E1 -2997.288,E2 -2997.288} C_VEL
LIN {X 0,Y 559.646,Z 240.45,A -85,B 0,C 180,E1 -3000.154,E2 -3000.154} C_VEL
LIN {X 0,Y 559.774,Z 232.324,A -85,B 0,C 180,E1 -3002.734,E2 -3002.734} C_VEL
LIN {X 0,Y 559.873,Z 224.411,A -85,B 0,C 180,E1 -3005.32,E2 -3005.32} C_VEL
LIN {X 0,Y 559.227,Z 219.239,A -85,B 0,C 180,E1 -3007.102,E2 -3007.102} C_VEL
LIN {X 0,Y 559.156,Z 218.837,A -85,B 0,C 180,E1 -3007.302,E2 -3007.302} C_VEL
LIN {X 0,Y 559.162,Z 218.836,A -85,B 0,C 180,E1 -3009.942,E2 -3009.942} C_VEL
LIN {X 0,Y 559.161,Z 218.832,A -85,B 0,C 180,E1 -3012.744,E2 -3012.744} C_VEL
LIN {X 0,Y 559.151,Z 218.835,A -85,B 0,C 180,E1 -3015.762,E2 -3015.762} C_VEL
LIN {X 0,Y 559.122,Z 218.836,A -85,B 0,C 180,E1 -3018.226,E2 -3018.226} C_VEL
LIN {X 0,Y 559.169,Z 218.83,A -85,B 0,C 180,E1 -3021.193,E2 -3021.193} C_VEL
LIN {X 0,Y 559.125,Z 218.84,A -85,B 0,C 180,E1 -3023.788,E2 -3023.788} C_VEL
LIN {X 0,Y 559.167,Z 218.831,A -85,B 0,C 180,E1 -3026.425,E2 -3026.425} C_VEL
LIN {X 0,Y 559.155,Z 218.838,A -85,B 0,C 180,E1 -3028.981,E2 -3028.981} C_VEL
LIN {X 0,Y 559.116,Z 218.836,A -85,B 0,C 180,E1 -3031.63,E2 -3031.63} C_VEL
LIN {X 0,Y 559.152,Z 218.834,A -85,B 0,C 180,E1 -3033.901,E2 -3033.901} C_VEL
LIN {X 0,Y 559.123,Z 218.836,A -85,B 0,C 180,E1 -3037.067,E2 -3037.067} C_VEL
LIN {X 0,Y 559.182,Z 218.834,A -85,B 0,C 180,E1 -3039.396,E2 -3039.396} C_VEL
LIN {X 0,Y 559.147,Z 218.834,A -85,B 0,C 180,E1 -3041.686,E2 -3041.686} C_VEL
LIN {X 0,Y 559.162,Z 218.832,A -85,B 0,C 180,E1 -3043.948,E2 -3043.948} C_VEL
LIN {X 0,Y 559.157,Z 218.838,A -85,B 0,C 180,E1 -3046.184,E2 -3046.184} C_VEL
LIN {X 0,Y 559.16,Z 218.832,A -85,B 0,C 180,E1 -3049.133,E2 -3049.133} C_VEL
LIN {X 0,Y 559.183,Z 218.828,A -85,B 0,C 180,E1 -3052.053,E2 -3052.053} C_VEL
LIN {X 0,Y 559.257,Z 218.824,A -85,B 0,C 180,E1 -3054.953,E2 -3054.953} C_VEL
LIN {X 0,Y 559.257,Z 218.822,A -85,B 0,C 180,E1 -3057.839,E2 -3057.839} C_VEL
LIN {X 0,Y 559.255,Z 218.824,A -85,B 0,C 180,E1 -3060,E2 -3060} C_VEL
LIN {X 0,Y 559.223,Z 218.824,A -85,B 0,C 180,E1 -3062.882,E2 -3062.882} C_VEL
LIN {X 0,Y 559.225,Z 218.823,A -85,B 0,C 180,E1 -3065.77,E2 -3065.77} C_VEL
LIN {X 0,Y 559.172,Z 218.834,A -85,B 0,C 180,E1 -3068.675,E2 -3068.675} C_VEL
LIN {X 0,Y 559.211,Z 218.829,A -85,B 0,C 180,E1 -3071.6,E2 -3071.6} C_VEL
LIN {X 0,Y 559.158,Z 218.832,A -85,B 0,C 180,E1 -3074.576,E2 -3074.576} C_VEL
LIN {X 0,Y 559.126,Z 218.835,A -85,B 0,C 180,E1 -3077.558,E2 -3077.558} C_VEL
LIN {X 0,Y 559.17,Z 218.831,A -85,B 0,C 180,E1 -3079.838,E2 -3079.838} C_VEL
LIN {X 0,Y 559.146,Z 218.839,A -85,B 0,C 180,E1 -3082.153,E2 -3082.153} C_VEL
LIN {X 0,Y 559.181,Z 218.833,A -85,B 0,C 180,E1 -3085.298,E2 -3085.298} C_VEL
LIN {X 0,Y 559.115,Z 218.838,A -85,B 0,C 180,E1 -3087.716,E2 -3087.716} C_VEL
LIN {X 0,Y 559.112,Z 218.837,A -85,B 0,C 180,E1 -3090.603,E2 -3090.603} C_VEL
LIN {X 0,Y 558.471,Z 218.919,A -85,B 0,C 180,E1 -3091.205,E2 -3091.205} C_VEL
LIN {X 0,Y 555.619,Z 219.276,A -85,B 0,C 180,E1 -3092.181,E2 -3092.181} C_VEL
LIN {X 0,Y 553.203,Z 219.574,A -85,B 0,C 180,E1 -3092.967,E2 -3092.967} C_VEL
LIN {X 0,Y 552.18,Z 219.702,A -85,B 0,C 180,E1 -3093.574,E2 -3093.574} C_VEL
LIN {X 0,Y 552.105,Z 219.712,A -85,B 0,C 180,E1 -3093.78,E2 -3093.78} C_VEL
LIN {X 0,Y 552.11,Z 219.71,A -85,B 0,C 180,E1 -3096.747,E2 -3096.747} C_VEL
LIN {X 0,Y 552.133,Z 219.71,A -85,B 0,C 180,E1 -3099.527,E2 -3099.527} C_VEL
LIN {X 0,Y 552.113,Z 219.714,A -85,B 0,C 180,E1 -3102.427,E2 -3102.427} C_VEL
LIN {X 0,Y 552.078,Z 219.714,A -85,B 0,C 180,E1 -3105.56,E2 -3105.56} C_VEL
LIN {X 0,Y 552.114,Z 219.709,A -85,B 0,C 180,E1 -3108.553,E2 -3108.553} C_VEL
LIN {X 0,Y 552.122,Z 219.712,A -85,B 0,C 180,E1 -3111.411,E2 -3111.411} C_VEL
LIN {X 0,Y 552.058,Z 219.718,A -85,B 0,C 180,E1 -3114.154,E2 -3114.154} C_VEL
LIN {X 0,Y 551.933,Z 219.878,A -85,B 0,C 180,E1 -3115.925,E2 -3115.925} C_VEL
LIN {X 0,Y 551.88,Z 222.74,A -85,B 0,C 180,E1 -3118.564,E2 -3118.564} C_VEL
LIN {X 0,Y 551.865,Z 225.427,A -85,B 0,C 180,E1 -3121.057,E2 -3121.057} C_VEL
LIN {X 0,Y 551.832,Z 228.115,A -85,B 0,C 180,E1 -3123.528,E2 -3123.528} C_VEL
LIN {X 0,Y 551.797,Z 230.82,A -85,B 0,C 180,E1 -3125.947,E2 -3125.947} C_VEL
LIN {X 0,Y 551.746,Z 234.378,A -85,B 0,C 180,E1 -3129.105,E2 -3129.105} C_VEL
LIN {X 0,Y 551.697,Z 237.073,A -85,B 0,C 180,E1 -3131.429,E2 -3131.429} C_VEL
LIN {X 0,Y 551.695,Z 239.713,A -85,B 0,C 180,E1 -3133.724,E2 -3133.724} C_VEL
LIN {X 0,Y 551.696,Z 242.343,A -85,B 0,C 180,E1 -3135.993,E2 -3135.993} C_VEL
LIN {X 0,Y 551.672,Z 243.672,A -85,B 0,C 180,E1 -3137.095,E2 -3137.095} C_VEL
LIN {X 0,Y 553.037,Z 252.23,A -85,B 0,C 180,E1 -3137.337,E2 -3137.337} C_VEL
LIN {X 0,Y 552.886,Z 265.006,A -85,B 0,C 180,E1 -3137.753,E2 -3137.753} C_VEL
LIN {X 0,Y 552.724,Z 277.639,A -85,B 0,C 180,E1 -3138.331,E2 -3138.331} C_VEL
LIN {X 0,Y 552.531,Z 288.905,A -85,B 0,C 180,E1 -3139.001,E2 -3139.001} C_VEL
LIN {X 0,Y 552.3,Z 299.945,A -85,B 0,C 180,E1 -3139.83,E2 -3139.83} C_VEL
LIN {X 0,Y 552.153,Z 310.679,A -85,B 0,C 180,E1 -3140.845,E2 -3140.845} C_VEL
LIN {X 0,Y 552.007,Z 318.598,A -85,B 0,C 180,E1 -3141.765,E2 -3141.765} C_VEL
LIN {X 0,Y 551.895,Z 326.459,A -85,B 0,C 180,E1 -3142.886,E2 -3142.886} C_VEL
LIN {X 0,Y 551.868,Z 333.456,A -85,B 0,C 180,E1 -3144.152,E2 -3144.152} C_VEL
LIN {X 0,Y 551.725,Z 338.197,A -85,B 0,C 180,E1 -3145.25,E2 -3145.25} C_VEL
LIN {X 0,Y 551.75,Z 341.829,A -85,B 0,C 180,E1 -3146.348,E2 -3146.348} C_VEL
LIN {X 0,Y 551.723,Z 343.706,A -85,B 0,C 180,E1 -3147.079,E2 -3147.079} C_VEL
LIN {X 0,Y 551.656,Z 345.128,A -85,B 0,C 180,E1 -3147.81,E2 -3147.81} C_VEL
LIN {X 0,Y 551.642,Z 346.757,A -85,B 0,C 180,E1 -3149.27,E2 -3149.27} C_VEL
LIN {X 0,Y 551.641,Z 346.996,A -85,B 0,C 180,E1 -3150,E2 -3150} C_VEL
LIN {X 0,Y 551.641,Z 346.815,A -85,B 0,C 180,E1 -3150.73,E2 -3150.73} C_VEL
LIN {X 0,Y 551.655,Z 345.264,A -85,B 0,C 180,E1 -3152.19,E2 -3152.19} C_VEL
LIN {X 0,Y 551.724,Z 343.903,A -85,B 0,C 180,E1 -3152.921,E2 -3152.921} C_VEL
LIN {X 0,Y 551.764,Z 341.026,A -85,B 0,C 180,E1 -3154.017,E2 -3154.017} C_VEL
LIN {X 0,Y 551.723,Z 337.125,A -85,B 0,C 180,E1 -3155.116,E2 -3155.116} C_VEL
LIN {X 0,Y 551.811,Z 331.394,A -85,B 0,C 180,E1 -3156.349,E2 -3156.349} C_VEL
LIN {X 0,Y 551.925,Z 324.537,A -85,B 0,C 180,E1 -3157.5,E2 -3157.5} C_VEL
LIN {X 0,Y 552.063,Z 316.355,A -85,B 0,C 180,E1 -3158.603,E2 -3158.603} C_VEL
LIN {X 0,Y 552.197,Z 307.986,A -85,B 0,C 180,E1 -3159.524,E2 -3159.524} C_VEL
LIN {X 0,Y 552.389,Z 297.663,A -85,B 0,C 180,E1 -3160.446,E2 -3160.446} C_VEL
LIN {X 0,Y 552.555,Z 286.937,A -85,B 0,C 180,E1 -3161.217,E2 -3161.217} C_VEL
LIN {X 0,Y 552.743,Z 276.26,A -85,B 0,C 180,E1 -3161.831,E2 -3161.831} C_VEL
LIN {X 0,Y 552.923,Z 263.73,A -85,B 0,C 180,E1 -3162.386,E2 -3162.386} C_VEL
LIN {X 0,Y 552.904,Z 250.743,A -85,B 0,C 180,E1 -3162.794,E2 -3162.794} C_VEL
LIN {X 0,Y 551.67,Z 243.668,A -85,B 0,C 180,E1 -3162.999,E2 -3162.999} C_VEL
LIN {X 0,Y 551.684,Z 240.73,A -85,B 0,C 180,E1 -3165.517,E2 -3165.517} C_VEL
LIN {X 0,Y 551.712,Z 238.062,A -85,B 0,C 180,E1 -3167.802,E2 -3167.802} C_VEL
LIN {X 0,Y 551.748,Z 235.395,A -85,B 0,C 180,E1 -3170.116,E2 -3170.116} C_VEL
LIN {X 0,Y 551.743,Z 232.694,A -85,B 0,C 180,E1 -3172.466,E2 -3172.466} C_VEL
LIN {X 0,Y 551.836,Z 229.532,A -85,B 0,C 180,E1 -3175.279,E2 -3175.279} C_VEL
LIN {X 0,Y 551.871,Z 226.418,A -85,B 0,C 180,E1 -3178.112,E2 -3178.112} C_VEL
LIN {X 0,Y 551.896,Z 223.72,A -85,B 0,C 180,E1 -3180.622,E2 -3180.622} C_VEL
LIN {X 0,Y 551.907,Z 220.945,A -85,B 0,C 180,E1 -3183.2,E2 -3183.2} C_VEL
LIN {X 0,Y 551.921,Z 219.91,A -85,B 0,C 180,E1 -3184.137,E2 -3184.137} C_VEL
LIN {X 0,Y 552.105,Z 219.712,A -85,B 0,C 180,E1 -3186.747,E2 -3186.747} C_VEL
LIN {X 0,Y 552.134,Z 219.707,A -85,B 0,C 180,E1 -3189.527,E2 -3189.527} C_VEL
LIN {X 0,Y 552.112,Z 219.714,A -85,B 0,C 180,E1 -3192.427,E2 -3192.427} C_VEL
LIN {X 0,Y 552.077,Z 219.717,A -85,B 0,C 180,E1 -3195.56,E2 -3195.56} C_VEL
LIN {X 0,Y 552.112,Z 219.71,A -85,B 0,C 180,E1 -3198.553,E2 -3198.553} C_VEL
LIN {X 0,Y 552.119,Z 219.71,A -85,B 0,C 180,E1 -3201.411,E2 -3201.411} C_VEL
LIN {X 0,Y 552.089,Z 219.718,A -85,B 0,C 180,E1 -3204.156,E2 -3204.156} C_VEL
LIN {X 0,Y 552.11,Z 219.709,A -85,B 0,C 180,E1 -3206.814,E2 -3206.814} C_VEL
LIN {X 0,Y 552.09,Z 219.718,A -85,B 0,C 180,E1 -3209.39,E2 -3209.39} C_VEL
LIN {X 0,Y 552.064,Z 219.715,A -85,B 0,C 180,E1 -3211.899,E2 -3211.899} C_VEL
LIN {X 0,Y 552.141,Z 219.711,A -85,B 0,C 180,E1 -3214.654,E2 -3214.654} C_VEL
LIN {X 0,Y 552.097,Z 219.714,A -85,B 0,C 180,E1 -3217.549,E2 -3217.549} C_VEL
LIN {X 0,Y 552.148,Z 219.705,A -85,B 0,C 180,E1 -3220.375,E2 -3220.375} C_VEL
LIN {X 0,Y 552.109,Z 219.714,A -85,B 0,C 180,E1 -3222.976,E2 -3222.976} C_VEL
LIN {X 0,Y 552.109,Z 219.711,A -85,B 0,C 180,E1 -3226.004,E2 -3226.004} C_VEL
LIN {X 0,Y 552.165,Z 219.703,A -85,B 0,C 180,E1 -3228.993,E2 -3228.993} C_VEL
LIN {X 0,Y 552.154,Z 219.707,A -85,B 0,C 180,E1 -3231.951,E2 -3231.951} C_VEL
LIN {X 0,Y 552.222,Z 219.701,A -85,B 0,C 180,E1 -3234.889,E2 -3234.889} C_VEL
LIN {X 0,Y 552.207,Z 219.697,A -85,B 0,C 180,E1 -3237.812,E2 -3237.812} C_VEL
LIN {X 0,Y 552.241,Z 219.694,A -85,B 0,C 180,E1 -3240.729,E2 -3240.729} C_VEL
LIN {X 0,Y 552.206,Z 219.698,A -85,B 0,C 180,E1 -3242.918,E2 -3242.918} C_VEL
LIN {X 0,Y 552.2,Z 219.7,A -85,B 0,C 180,E1 -3245.844,E2 -3245.844} C_VEL
LIN {X 0,Y 552.137,Z 219.711,A -85,B 0,C 180,E1 -3248.786,E2 -3248.786} C_VEL
LIN {X 0,Y 552.103,Z 219.712,A -85,B 0,C 180,E1 -3251.752,E2 -3251.752} C_VEL
LIN {X 0,Y 552.132,Z 219.707,A -85,B 0,C 180,E1 -3254.749,E2 -3254.749} C_VEL
LIN {X 0,Y 552.113,Z 219.711,A -85,B 0,C 180,E1 -3257.788,E2 -3257.788} C_VEL
LIN {X 0,Y 552.131,Z 219.708,A -85,B 0,C 180,E1 -3260.101,E2 -3260.101} C_VEL
LIN {X 0,Y 552.094,Z 219.716,A -85,B 0,C 180,E1 -3262.451,E2 -3262.451} C_VEL
LIN {X 0,Y 552.082,Z 219.714,A -85,B 0,C 180,E1 -3265.333,E2 -3265.333} C_VEL
LIN {X 0,Y 552.058,Z 219.716,A -85,B 0,C 180,E1 -3268.101,E2 -3268.101} C_VEL
LIN {X 0,Y 552.098,Z 219.714,A -85,B 0,C 180,E1 -3270.61,E2 -3270.61} C_VEL
LIN {X 0,Y 552.119,Z 219.71,A -85,B 0,C 180,E1 -3273.186,E2 -3273.186} C_VEL
LIN {X 0,Y 552.077,Z 219.718,A -85,B 0,C 180,E1 -3275.844,E2 -3275.844} C_VEL
LIN {X 0,Y 552.113,Z 219.709,A -85,B 0,C 180,E1 -3278.589,E2 -3278.589} C_VEL
LIN {X 0,Y 552.075,Z 219.717,A -85,B 0,C 180,E1 -3281.45,E2 -3281.45} C_VEL
LIN {X 0,Y 552.094,Z 219.717,A -85,B 0,C 180,E1 -3284.438,E2 -3284.438} C_VEL
LIN {X 0,Y 552.132,Z 219.71,A -85,B 0,C 180,E1 -3287.585,E2 -3287.585} C_VEL
LIN {X 0,Y 552.13,Z 219.71,A -85,B 0,C 180,E1 -3290.473,E2 -3290.473} C_VEL
LIN {X 0,Y 552.13,Z 219.844,A -85,B 0,C 180,E1 -3292.569,E2 -3292.569} C_VEL
LIN {X 0,Y 552.911,Z 225.193,A -85,B 0,C 180,E1 -3294.439,E2 -3294.439} C_VEL
LIN {X 0,Y 552.843,Z 233.038,A -85,B 0,C 180,E1 -3297.037,E2 -3297.037} C_VEL
LIN {X 0,Y 552.661,Z 241.792,A -85,B 0,C 180,E1 -3299.852,E2 -3299.852} C_VEL
LIN {X 0,Y 552.52,Z 251.611,A -85,B 0,C 180,E1 -3302.923,E2 -3302.923} C_VEL
LIN {X 0,Y 552.353,Z 261.633,A -85,B 0,C 180,E1 -3305.973,E2 -3305.973} C_VEL
LIN {X 0,Y 552.2,Z 270.901,A -85,B 0,C 180,E1 -3308.732,E2 -3308.732} C_VEL
LIN {X 0,Y 552.084,Z 280.168,A -85,B 0,C 180,E1 -3311.443,E2 -3311.443} C_VEL
LIN {X 0,Y 551.976,Z 290.759,A -85,B 0,C 180,E1 -3314.492,E2 -3314.492} C_VEL
LIN {X 0,Y 551.883,Z 299.53,A -85,B 0,C 180,E1 -3316.983,E2 -3316.983} C_VEL
LIN {X 0,Y 553.097,Z 308.523,A -85,B 0,C 180,E1 -3317.199,E2 -3317.199} C_VEL
LIN {X 0,Y 552.949,Z 321.178,A -85,B 0,C 180,E1 -3317.568,E2 -3317.568} C_VEL
LIN {X 0,Y 552.743,Z 333.486,A -85,B 0,C 180,E1 -3318.076,E2 -3318.076} C_VEL
LIN {X 0,Y 552.56,Z 345.389,A -85,B 0,C 180,E1 -3318.727,E2 -3318.727} C_VEL
LIN {X 0,Y 552.385,Z 357.097,A -85,B 0,C 180,E1 -3319.554,E2 -3319.554} C_VEL
LIN {X 0,Y 552.201,Z 367.538,A -85,B 0,C 180,E1 -3320.476,E2 -3320.476} C_VEL
LIN {X 0,Y 552.082,Z 375.991,A -85,B 0,C 180,E1 -3321.398,E2 -3321.398} C_VEL
LIN {X 0,Y 551.926,Z 384.238,A -85,B 0,C 180,E1 -3322.5,E2 -3322.5} C_VEL
LIN {X 0,Y 551.821,Z 391.209,A -85,B 0,C 180,E1 -3323.662,E2 -3323.662} C_VEL
LIN {X 0,Y 551.723,Z 396.95,A -85,B 0,C 180,E1 -3324.884,E2 -3324.884} C_VEL
LIN {X 0,Y 551.764,Z 400.896,A -85,B 0,C 180,E1 -3325.983,E2 -3325.983} C_VEL
LIN {X 0,Y 551.723,Z 403.809,A -85,B 0,C 180,E1 -3327.079,E2 -3327.079} C_VEL
LIN {X 0,Y 551.645,Z 406.185,A -85,B 0,C 180,E1 -3328.54,E2 -3328.54} C_VEL
LIN {X 0,Y 551.64,Z 407,A -85,B 0,C 180,E1 -3330,E2 -3330} C_VEL
LIN {X 0,Y 551.645,Z 406.186,A -85,B 0,C 180,E1 -3331.46,E2 -3331.46} C_VEL
LIN {X 0,Y 551.657,Z 405.2,A -85,B 0,C 180,E1 -3332.19,E2 -3332.19} C_VEL
LIN {X 0,Y 551.723,Z 403.809,A -85,B 0,C 180,E1 -3332.921,E2 -3332.921} C_VEL
LIN {X 0,Y 551.764,Z 400.895,A -85,B 0,C 180,E1 -3334.017,E2 -3334.017} C_VEL
LIN {X 0,Y 551.724,Z 396.949,A -85,B 0,C 180,E1 -3335.116,E2 -3335.116} C_VEL
LIN {X 0,Y 551.825,Z 391.189,A -85,B 0,C 180,E1 -3336.341,E2 -3336.341} C_VEL
LIN {X 0,Y 551.927,Z 384.236,A -85,B 0,C 180,E1 -3337.5,E2 -3337.5} C_VEL
LIN {X 0,Y 552.082,Z 375.989,A -85,B 0,C 180,E1 -3338.603,E2 -3338.603} C_VEL
LIN {X 0,Y 552.201,Z 367.536,A -85,B 0,C 180,E1 -3339.524,E2 -3339.524} C_VEL
LIN {X 0,Y 552.385,Z 357.094,A -85,B 0,C 180,E1 -3340.446,E2 -3340.446} C_VEL
LIN {X 0,Y 552.565,Z 345.348,A -85,B 0,C 180,E1 -3341.276,E2 -3341.276} C_VEL
LIN {X 0,Y 552.742,Z 333.48,A -85,B 0,C 180,E1 -3341.924,E2 -3341.924} C_VEL
LIN {X 0,Y 552.949,Z 321.167,A -85,B 0,C 180,E1 -3342.432,E2 -3342.432} C_VEL
LIN {X 0,Y 553.097,Z 308.512,A -85,B 0,C 180,E1 -3342.802,E2 -3342.802} C_VEL
LIN {X 0,Y 552.033,Z 300.752,A -85,B 0,C 180,E1 -3342.98,E2 -3342.98} C_VEL
LIN {X 0,Y 551.883,Z 299.529,A -85,B 0,C 180,E1 -3343.017,E2 -3343.017} C_VEL
LIN {X 0,Y 551.99,Z 289.435,A -85,B 0,C 180,E1 -3345.887,E2 -3345.887} C_VEL
LIN {X 0,Y 552.082,Z 278.843,A -85,B 0,C 180,E1 -3348.942,E2 -3348.942} C_VEL
LIN {X 0,Y 552.254,Z 268.253,A -85,B 0,C 180,E1 -3352.05,E2 -3352.05} C_VEL
LIN {X 0,Y 552.381,Z 258.985,A -85,B 0,C 180,E1 -3354.826,E2 -3354.826} C_VEL
LIN {X 0,Y 552.531,Z 249.717,A -85,B 0,C 180,E1 -3357.663,E2 -3357.663} C_VEL
LIN {X 0,Y 552.681,Z 240.45,A -85,B 0,C 180,E1 -3360.574,E2 -3360.574} C_VEL
LIN {X 0,Y 552.855,Z 232.507,A -85,B 0,C 180,E1 -3363.136,E2 -3363.136} C_VEL
LIN {X 0,Y 552.915,Z 225.191,A -85,B 0,C 180,E1 -3365.561,E2 -3365.561} C_VEL
LIN {X 0,Y 552.12,Z 219.714,A -85,B 0,C 180,E1 -3367.489,E2 -3367.489} C_VEL
LIN {X 0,Y 552.112,Z 219.715,A -85,B 0,C 180,E1 -3370.481,E2 -3370.481} C_VEL
LIN {X 0,Y 552.111,Z 219.714,A -85,B 0,C 180,E1 -3373.424,E2 -3373.424} C_VEL
LIN {X 0,Y 552.111,Z 219.71,A -85,B 0,C 180,E1 -3376.576,E2 -3376.576} C_VEL
LIN {X 0,Y 552.099,Z 219.71,A -85,B 0,C 180,E1 -3379.799,E2 -3379.799} C_VEL
LIN {X 0,Y 552.088,Z 219.719,A -85,B 0,C 180,E1 -3382.336,E2 -3382.336} C_VEL
LIN {X 0,Y 552.086,Z 219.713,A -85,B 0,C 180,E1 -3385.051,E2 -3385.051} C_VEL
LIN {X 0,Y 552.12,Z 219.712,A -85,B 0,C 180,E1 -3387.682,E2 -3387.682} C_VEL
LIN {X 0,Y 552.09,Z 219.713,A -85,B 0,C 180,E1 -3390.234,E2 -3390.234} C_VEL
LIN {X 0,Y 552.082,Z 219.713,A -85,B 0,C 180,E1 -3393.013,E2 -3393.013} C_VEL
LIN {X 0,Y 552.08,Z 219.72,A -85,B 0,C 180,E1 -3395.961,E2 -3395.961} C_VEL
LIN {X 0,Y 552.131,Z 219.707,A -85,B 0,C 180,E1 -3398.338,E2 -3398.338} C_VEL
LIN {X 0,Y 552.157,Z 219.706,A -85,B 0,C 180,E1 -3400.674,E2 -3400.674} C_VEL
LIN {X 0,Y 552.114,Z 219.709,A -85,B 0,C 180,E1 -3403.737,E2 -3403.737} C_VEL
LIN {X 0,Y 552.127,Z 219.712,A -85,B 0,C 180,E1 -3406.004,E2 -3406.004} C_VEL
LIN {X 0,Y 552.129,Z 219.707,A -85,B 0,C 180,E1 -3408.993,E2 -3408.993} C_VEL
LIN {X 0,Y 552.141,Z 219.706,A -85,B 0,C 180,E1 -3411.951,E2 -3411.951} C_VEL
LIN {X 0,Y 552.232,Z 219.7,A -85,B 0,C 180,E1 -3414.889,E2 -3414.889} C_VEL
LIN {X 0,Y 552.229,Z 219.698,A -85,B 0,C 180,E1 -3417.812,E2 -3417.812} C_VEL
LIN {X 0,Y 552.224,Z 219.7,A -85,B 0,C 180,E1 -3420,E2 -3420} C_VEL
LIN {X 0,Y 552.191,Z 219.701,A -85,B 0,C 180,E1 -3422.918,E2 -3422.918} C_VEL
LIN {X 0,Y 552.195,Z 219.699,A -85,B 0,C 180,E1 -3425.844,E2 -3425.844} C_VEL
LIN {X 0,Y 552.145,Z 219.708,A -85,B 0,C 180,E1 -3428.786,E2 -3428.786} C_VEL
LIN {X 0,Y 552.167,Z 219.708,A -85,B 0,C 180,E1 -3431.75,E2 -3431.75} C_VEL
LIN {X 0,Y 552.125,Z 219.709,A -85,B 0,C 180,E1 -3434.749,E2 -3434.749} C_VEL
LIN {X 0,Y 552.088,Z 219.711,A -85,B 0,C 180,E1 -3437.789,E2 -3437.789} C_VEL
LIN {X 0,Y 552.131,Z 219.71,A -85,B 0,C 180,E1 -3440.101,E2 -3440.101} C_VEL
LIN {X 0,Y 552.097,Z 219.714,A -85,B 0,C 180,E1 -3442.451,E2 -3442.451} C_VEL
LIN {X 0,Y 552.143,Z 219.711,A -85,B 0,C 180,E1 -3445.346,E2 -3445.346} C_VEL
LIN {X 0,Y 552.063,Z 219.715,A -85,B 0,C 180,E1 -3448.101,E2 -3448.101} C_VEL
LIN {X 0,Y 552.08,Z 219.72,A -85,B 0,C 180,E1 -3450.611,E2 -3450.611} C_VEL
LIN {X 0,Y 552.111,Z 219.709,A -85,B 0,C 180,E1 -3453.186,E2 -3453.186} C_VEL
LIN {X 0,Y 552.105,Z 219.712,A -85,B 0,C 180,E1 -3453.78,E2 -3453.78} C_VEL
LIN {X 0,Y 551.471,Z 219.795,A -85,B 0,C 180,E1 -3454.388,E2 -3454.388} C_VEL
LIN {X 0,Y 548.654,Z 220.144,A -85,B 0,C 180,E1 -3455.377,E2 -3455.377} C_VEL
LIN {X 0,Y 546.237,Z 220.444,A -85,B 0,C 180,E1 -3456.172,E2 -3456.172} C_VEL
LIN {X 0,Y 545.169,Z 220.575,A -85,B 0,C 180,E1 -3456.786,E2 -3456.786} C_VEL
LIN {X 0,Y 545.067,Z 220.589,A -85,B 0,C 180,E1 -3456.994,E2 -3456.994} C_VEL
LIN {X 0,Y 545.069,Z 220.587,A -85,B 0,C 180,E1 -3460.143,E2 -3460.143} C_VEL
LIN {X 0,Y 545.042,Z 220.595,A -85,B 0,C 180,E1 -3462.694,E2 -3462.694} C_VEL
LIN {X 0,Y 545.025,Z 220.591,A -85,B 0,C 180,E1 -3465.171,E2 -3465.171} C_VEL
LIN {X 0,Y 545.073,Z 220.586,A -85,B 0,C 180,E1 -3468.403,E2 -3468.403} C_VEL
LIN {X 0,Y 545.085,Z 220.588,A -85,B 0,C 180,E1 -3470.818,E2 -3470.818} C_VEL
LIN {X 0,Y 545.034,Z 220.592,A -85,B 0,C 180,E1 -3473.619,E2 -3473.619} C_VEL
LIN {X 0,Y 544.878,Z 220.617,A -85,B 0,C 180,E1 -3475.639,E2 -3475.639} C_VEL
LIN {X 0,Y 544.831,Z 221.704,A -85,B 0,C 180,E1 -3476.978,E2 -3476.978} C_VEL
LIN {X 0,Y 544.843,Z 224.718,A -85,B 0,C 180,E1 -3479.797,E2 -3479.797} C_VEL
LIN {X 0,Y 544.783,Z 228.053,A -85,B 0,C 180,E1 -3482.891,E2 -3482.891} C_VEL
LIN {X 0,Y 544.734,Z 231.041,A -85,B 0,C 180,E1 -3485.615,E2 -3485.615} C_VEL
LIN {X 0,Y 544.676,Z 234.657,A -85,B 0,C 180,E1 -3488.821,E2 -3488.821} C_VEL
LIN {X 0,Y 544.635,Z 237.363,A -85,B 0,C 180,E1 -3491.179,E2 -3491.179} C_VEL
LIN {X 0,Y 544.649,Z 240.06,A -85,B 0,C 180,E1 -3493.508,E2 -3493.508} C_VEL
LIN {X 0,Y 544.623,Z 242.708,A -85,B 0,C 180,E1 -3495.807,E2 -3495.807} C_VEL
LIN {X 0,Y 544.59,Z 243.995,A -85,B 0,C 180,E1 -3496.924,E2 -3496.924} C_VEL
LIN {X 0,Y 546.125,Z 253.401,A -85,B 0,C 180,E1 -3497.198,E2 -3497.198} C_VEL
LIN {X 0,Y 545.953,Z 266.346,A -85,B 0,C 180,E1 -3497.642,E2 -3497.642} C_VEL
LIN {X 0,Y 545.779,Z 278.428,A -85,B 0,C 180,E1 -3498.215,E2 -3498.215} C_VEL
LIN {X 0,Y 545.55,Z 288.999,A -85,B 0,C 180,E1 -3498.858,E2 -3498.858} C_VEL
LIN {X 0,Y 545.312,Z 299.965,A -85,B 0,C 180,E1 -3499.699,E2 -3499.699} C_VEL
LIN {X 0,Y 545.123,Z 310.684,A -85,B 0,C 180,E1 -3500.726,E2 -3500.726} C_VEL
LIN {X 0,Y 544.975,Z 318.603,A -85,B 0,C 180,E1 -3501.658,E2 -3501.658} C_VEL
LIN {X 0,Y 544.83,Z 326.351,A -85,B 0,C 180,E1 -3502.775,E2 -3502.775} C_VEL
LIN {X 0,Y 544.778,Z 333.459,A -85,B 0,C 180,E1 -3504.076,E2 -3504.076} C_VEL
LIN {X 0,Y 544.629,Z 338.199,A -85,B 0,C 180,E1 -3505.188,E2 -3505.188} C_VEL
LIN {X 0,Y 544.669,Z 341.831,A -85,B 0,C 180,E1 -3506.301,E2 -3506.301} C_VEL
LIN {X 0,Y 544.65,Z 343.708,A -85,B 0,C 180,E1 -3507.041,E2 -3507.041} C_VEL
LIN {X 0,Y 544.57,Z 345.128,A -85,B 0,C 180,E1 -3507.781,E2 -3507.781} C_VEL
LIN {X 0,Y 544.542,Z 346.757,A -85,B 0,C 180,E1 -3509.26,E2 -3509.26} C_VEL
LIN {X 0,Y 544.541,Z 346.996,A -85,B 0,C 180,E1 -3510,E2 -3510} C_VEL
LIN {X 0,Y 544.542,Z 346.815,A -85,B 0,C 180,E1 -3510.739,E2 -3510.739} C_VEL
LIN {X 0,Y 544.57,Z 345.262,A -85,B 0,C 180,E1 -3512.219,E2 -3512.219} C_VEL
LIN {X 0,Y 544.651,Z 343.901,A -85,B 0,C 180,E1 -3512.959,E2 -3512.959} C_VEL
LIN {X 0,Y 544.684,Z 341.024,A -85,B 0,C 180,E1 -3514.069,E2 -3514.069} C_VEL
LIN {X 0,Y 544.653,Z 337.122,A -85,B 0,C 180,E1 -3515.182,E2 -3515.182} C_VEL
LIN {X 0,Y 544.724,Z 331.898,A -85,B 0,C 180,E1 -3516.335,E2 -3516.335} C_VEL
LIN {X 0,Y 544.859,Z 324.532,A -85,B 0,C 180,E1 -3517.597,E2 -3517.597} C_VEL
LIN {X 0,Y 544.999,Z 316.35,A -85,B 0,C 180,E1 -3518.715,E2 -3518.715} C_VEL
LIN {X 0,Y 545.16,Z 307.98,A -85,B 0,C 180,E1 -3519.648,E2 -3519.648} C_VEL
LIN {X 0,Y 545.367,Z 297.684,A -85,B 0,C 180,E1 -3520.582,E2 -3520.582} C_VEL
LIN {X 0,Y 545.612,Z 286.303,A -85,B 0,C 180,E1 -3521.409,E2 -3521.409} C_VEL
LIN {X 0,Y 545.838,Z 274.598,A -85,B 0,C 180,E1 -3522.077,E2 -3522.077} C_VEL
LIN {X 0,Y 546.017,Z 262.623,A -85,B 0,C 180,E1 -3522.592,E2 -3522.592} C_VEL
LIN {X 0,Y 546.037,Z 251.884,A -85,B 0,C 180,E1 -3522.934,E2 -3522.934} C_VEL
LIN {X 0,Y 544.601,Z 244.016,A -85,B 0,C 180,E1 -3523.171,E2 -3523.171} C_VEL
LIN {X 0,Y 544.605,Z 241.054,A -85,B 0,C 180,E1 -3525.724,E2 -3525.724} C_VEL
LIN {X 0,Y 544.631,Z 238.384,A -85,B 0,C 180,E1 -3528.041,E2 -3528.041} C_VEL
LIN {X 0,Y 544.66,Z 235.661,A -85,B 0,C 180,E1 -3530.389,E2 -3530.389} C_VEL
LIN {X 0,Y 544.666,Z 232.943,A -85,B 0,C 180,E1 -3532.774,E2 -3532.774} C_VEL
LIN {X 0,Y 544.772,Z 229.968,A -85,B 0,C 180,E1 -3535.437,E2 -3535.437} C_VEL
LIN {X 0,Y 544.808,Z 226.638,A -85,B 0,C 180,E1 -3538.509,E2 -3538.509} C_VEL
LIN {X 0,Y 544.805,Z 223.91,A -85,B 0,C 180,E1 -3541.064,E2 -3541.064} C_VEL
LIN {X 0,Y 544.838,Z 221.096,A -85,B 0,C 180,E1 -3543.688,E2 -3543.688} C_VEL
LIN {X 0,Y 544.89,Z 220.615,A -85,B 0,C 180,E1 -3544.577,E2 -3544.577} C_VEL
LIN {X 0,Y 545.039,Z 220.595,A -85,B 0,C 180,E1 -3547.304,E2 -3547.304} C_VEL
LIN {X 0,Y 545.069,Z 220.588,A -85,B 0,C 180,E1 -3550.143,E2 -3550.143} C_VEL
LIN {X 0,Y 545.041,Z 220.592,A -85,B 0,C 180,E1 -3552.694,E2 -3552.694} C_VEL
LIN {X 0,Y 545.024,Z 220.592,A -85,B 0,C 180,E1 -3555.171,E2 -3555.171} C_VEL
LIN {X 0,Y 545.071,Z 220.587,A -85,B 0,C 180,E1 -3558.404,E2 -3558.404} C_VEL
LIN {X 0,Y 545.082,Z 220.59,A -85,B 0,C 180,E1 -3560.818,E2 -3560.818} C_VEL
LIN {X 0,Y 545.045,Z 220.59,A -85,B 0,C 180,E1 -3563.62,E2 -3563.62} C_VEL
LIN {X 0,Y 545.061,Z 220.59,A -85,B 0,C 180,E1 -3566.328,E2 -3566.328} C_VEL
LIN {X 0,Y 545.063,Z 220.588,A -85,B 0,C 180,E1 -3568.952,E2 -3568.952} C_VEL
LIN {X 0,Y 545.043,Z 220.592,A -85,B 0,C 180,E1 -3571.504,E2 -3571.504} C_VEL
LIN {X 0,Y 545.079,Z 220.587,A -85,B 0,C 180,E1 -3573.999,E2 -3573.999} C_VEL
LIN {X 0,Y 545.085,Z 220.59,A -85,B 0,C 180,E1 -3576.441,E2 -3576.441} C_VEL
LIN {X 0,Y 545.096,Z 220.589,A -85,B 0,C 180,E1 -3579.628,E2 -3579.628} C_VEL
LIN {X 0,Y 545.054,Z 220.59,A -85,B 0,C 180,E1 -3582.748,E2 -3582.748} C_VEL
LIN {X 0,Y 545.068,Z 220.587,A -85,B 0,C 180,E1 -3585.819,E2 -3585.819} C_VEL
LIN {X 0,Y 545.121,Z 220.581,A -85,B 0,C 180,E1 -3588.849,E2 -3588.849} C_VEL
LIN {X 0,Y 545.125,Z 220.584,A -85,B 0,C 180,E1 -3591.847,E2 -3591.847} C_VEL
LIN {X 0,Y 545.199,Z 220.575,A -85,B 0,C 180,E1 -3594.823,E2 -3594.823} C_VEL
LIN {X 0,Y 545.181,Z 220.572,A -85,B 0,C 180,E1 -3597.784,E2 -3597.784} C_VEL
LIN {X 0,Y 545.211,Z 220.57,A -85,B 0,C 180,E1 -3600.739,E2 -3600.739} C_VEL
LIN {X 0,Y 545.173,Z 220.575,A -85,B 0,C 180,E1 -3602.956,E2 -3602.956} C_VEL
LIN {X 0,Y 545.172,Z 220.575,A -85,B 0,C 180,E1 -3605.919,E2 -3605.919} C_VEL
LIN {X 0,Y 545.097,Z 220.587,A -85,B 0,C 180,E1 -3608.9,E2 -3608.9} C_VEL
LIN {X 0,Y 545.068,Z 220.59,A -85,B 0,C 180,E1 -3611.906,E2 -3611.906} C_VEL
LIN {X 0,Y 545.085,Z 220.585,A -85,B 0,C 180,E1 -3614.944,E2 -3614.944} C_VEL
LIN {X 0,Y 545.081,Z 220.586,A -85,B 0,C 180,E1 -3618.026,E2 -3618.026} C_VEL
LIN {X 0,Y 545.096,Z 220.587,A -85,B 0,C 180,E1 -3620.372,E2 -3620.372} C_VEL
LIN {X 0,Y 545.075,Z 220.587,A -85,B 0,C 180,E1 -3623.56,E2 -3623.56} C_VEL
LIN {X 0,Y 545.047,Z 220.589,A -85,B 0,C 180,E1 -3626.827,E2 -3626.827} C_VEL
LIN {X 0,Y 545.031,Z 220.597,A -85,B 0,C 180,E1 -3629.341,E2 -3629.341} C_VEL
LIN {X 0,Y 545.059,Z 220.589,A -85,B 0,C 180,E1 -3631.915,E2 -3631.915} C_VEL
LIN {X 0,Y 545.065,Z 220.592,A -85,B 0,C 180,E1 -3634.564,E2 -3634.564} C_VEL
LIN {X 0,Y 545.032,Z 220.593,A -85,B 0,C 180,E1 -3637.305,E2 -3637.305} C_VEL
LIN {X 0,Y 545.052,Z 220.588,A -85,B 0,C 180,E1 -3640.144,E2 -3640.144} C_VEL
LIN {X 0,Y 545.047,Z 220.593,A -85,B 0,C 180,E1 -3643.11,E2 -3643.11} C_VEL
LIN {X 0,Y 545.051,Z 220.595,A -85,B 0,C 180,E1 -3646.226,E2 -3646.226} C_VEL
LIN {X 0,Y 545.084,Z 220.586,A -85,B 0,C 180,E1 -3648.885,E2 -3648.885} C_VEL
LIN {X 0,Y 545.079,Z 220.589,A -85,B 0,C 180,E1 -3650.818,E2 -3650.818} C_VEL
LIN {X 0,Y 545.09,Z 220.73,A -85,B 0,C 180,E1 -3652.351,E2 -3652.351} C_VEL
LIN {X 0,Y 545.918,Z 225.96,A -85,B 0,C 180,E1 -3654.198,E2 -3654.198} C_VEL
LIN {X 0,Y 545.93,Z 232.49,A -85,B 0,C 180,E1 -3656.388,E2 -3656.388} C_VEL
LIN {X 0,Y 545.739,Z 240.451,A -85,B 0,C 180,E1 -3658.995,E2 -3658.995} C_VEL
LIN {X 0,Y 545.564,Z 249.718,A -85,B 0,C 180,E1 -3661.953,E2 -3661.953} C_VEL
LIN {X 0,Y 545.357,Z 258.986,A -85,B 0,C 180,E1 -3664.832,E2 -3664.832} C_VEL
LIN {X 0,Y 545.225,Z 268.253,A -85,B 0,C 180,E1 -3667.65,E2 -3667.65} C_VEL
LIN {X 0,Y 545.068,Z 278.844,A -85,B 0,C 180,E1 -3670.804,E2 -3670.804} C_VEL
LIN {X 0,Y 544.933,Z 289.435,A -85,B 0,C 180,E1 -3673.902,E2 -3673.902} C_VEL
LIN {X 0,Y 544.798,Z 299.53,A -85,B 0,C 180,E1 -3676.811,E2 -3676.811} C_VEL
LIN {X 0,Y 546.177,Z 309.438,A -85,B 0,C 180,E1 -3677.057,E2 -3677.057} C_VEL
LIN {X 0,Y 546.003,Z 322.475,A -85,B 0,C 180,E1 -3677.455,E2 -3677.455} C_VEL
LIN {X 0,Y 545.783,Z 333.487,A -85,B 0,C 180,E1 -3677.922,E2 -3677.922} C_VEL
LIN {X 0,Y 545.584,Z 344.156,A -85,B 0,C 180,E1 -3678.505,E2 -3678.505} C_VEL
LIN {X 0,Y 545.425,Z 354.747,A -85,B 0,C 180,E1 -3679.232,E2 -3679.232} C_VEL
LIN {X 0,Y 545.225,Z 365.602,A -85,B 0,C 180,E1 -3680.166,E2 -3680.166} C_VEL
LIN {X 0,Y 545.051,Z 374.413,A -85,B 0,C 180,E1 -3681.099,E2 -3681.099} C_VEL
LIN {X 0,Y 544.895,Z 383.001,A -85,B 0,C 180,E1 -3682.217,E2 -3682.217} C_VEL
LIN {X 0,Y 544.745,Z 390.35,A -85,B 0,C 180,E1 -3683.421,E2 -3683.421} C_VEL
LIN {X 0,Y 544.741,Z 395.366,A -85,B 0,C 180,E1 -3684.447,E2 -3684.447} C_VEL
LIN {X 0,Y 544.66,Z 399.678,A -85,B 0,C 180,E1 -3685.56,E2 -3685.56} C_VEL
LIN {X 0,Y 544.669,Z 401.957,A -85,B 0,C 180,E1 -3686.301,E2 -3686.301} C_VEL
LIN {X 0,Y 544.65,Z 403.808,A -85,B 0,C 180,E1 -3687.041,E2 -3687.041} C_VEL
LIN {X 0,Y 544.546,Z 406.186,A -85,B 0,C 180,E1 -3688.521,E2 -3688.521} C_VEL
LIN {X 0,Y 544.541,Z 407,A -85,B 0,C 180,E1 -3690,E2 -3690} C_VEL
LIN {X 0,Y 544.546,Z 406.186,A -85,B 0,C 180,E1 -3691.479,E2 -3691.479} C_VEL
LIN {X 0,Y 544.65,Z 403.81,A -85,B 0,C 180,E1 -3692.959,E2 -3692.959} C_VEL
LIN {X 0,Y 544.684,Z 400.895,A -85,B 0,C 180,E1 -3694.07,E2 -3694.07} C_VEL
LIN {X 0,Y 544.653,Z 396.948,A -85,B 0,C 180,E1 -3695.182,E2 -3695.182} C_VEL
LIN {X 0,Y 544.737,Z 391.595,A -85,B 0,C 180,E1 -3696.349,E2 -3696.349} C_VEL
LIN {X 0,Y 544.86,Z 384.236,A -85,B 0,C 180,E1 -3697.598,E2 -3697.598} C_VEL
LIN {X 0,Y 545.029,Z 375.989,A -85,B 0,C 180,E1 -3698.715,E2 -3698.715} C_VEL
LIN {X 0,Y 545.164,Z 367.536,A -85,B 0,C 180,E1 -3699.648,E2 -3699.648} C_VEL
LIN {X 0,Y 545.381,Z 357.095,A -85,B 0,C 180,E1 -3700.582,E2 -3700.582} C_VEL
LIN {X 0,Y 545.587,Z 345.661,A -85,B 0,C 180,E1 -3701.401,E2 -3701.401} C_VEL
LIN {X 0,Y 545.763,Z 335.407,A -85,B 0,C 180,E1 -3701.985,E2 -3701.985} C_VEL
LIN {X 0,Y 545.988,Z 323.758,A -85,B 0,C 180,E1 -3702.499,E2 -3702.499} C_VEL
LIN {X 0,Y 546.135,Z 310.341,A -85,B 0,C 180,E1 -3702.92,E2 -3702.92} C_VEL
LIN {X 0,Y 545.896,Z 306.358,A -85,B 0,C 180,E1 -3703.021,E2 -3703.021} C_VEL
LIN {X 0,Y 544.799,Z 299.529,A -85,B 0,C 180,E1 -3703.19,E2 -3703.19} C_VEL
LIN {X 0,Y 544.933,Z 289.435,A -85,B 0,C 180,E1 -3706.098,E2 -3706.098} C_VEL
LIN {X 0,Y 545.067,Z 278.843,A -85,B 0,C 180,E1 -3709.196,E2 -3709.196} C_VEL
LIN {X 0,Y 545.218,Z 268.252,A -85,B 0,C 180,E1 -3712.35,E2 -3712.35} C_VEL
LIN {X 0,Y 545.357,Z 258.985,A -85,B 0,C 180,E1 -3715.168,E2 -3715.168} C_VEL
LIN {X 0,Y 545.565,Z 249.717,A -85,B 0,C 180,E1 -3718.047,E2 -3718.047} C_VEL
LIN {X 0,Y 545.74,Z 240.45,A -85,B 0,C 180,E1 -3721.006,E2 -3721.006} C_VEL
LIN {X 0,Y 545.931,Z 232.489,A -85,B 0,C 180,E1 -3723.612,E2 -3723.612} C_VEL
LIN {X 0,Y 545.94,Z 225.952,A -85,B 0,C 180,E1 -3725.805,E2 -3725.805} C_VEL
LIN {X 0,Y 545.048,Z 220.595,A -85,B 0,C 180,E1 -3727.769,E2 -3727.769} C_VEL
LIN {X 0,Y 545.084,Z 220.591,A -85,B 0,C 180,E1 -3730.473,E2 -3730.473} C_VEL
LIN {X 0,Y 545.082,Z 220.587,A -85,B 0,C 180,E1 -3733.107,E2 -3733.107} C_VEL
LIN {X 0,Y 545.053,Z 220.589,A -85,B 0,C 180,E1 -3736.226,E2 -3736.226} C_VEL
LIN {X 0,Y 545.027,Z 220.597,A -85,B 0,C 180,E1 -3738.88,E2 -3738.88} C_VEL
LIN {X 0,Y 545.047,Z 220.59,A -85,B 0,C 180,E1 -3741.762,E2 -3741.762} C_VEL
LIN {X 0,Y 545.034,Z 220.592,A -85,B 0,C 180,E1 -3744.531,E2 -3744.531} C_VEL
LIN {X 0,Y 545.074,Z 220.591,A -85,B 0,C 180,E1 -3747.212,E2 -3747.212} C_VEL
LIN {X 0,Y 545.066,Z 220.587,A -85,B 0,C 180,E1 -3749.81,E2 -3749.81} C_VEL
LIN {X 0,Y 545.029,Z 220.593,A -85,B 0,C 180,E1 -3752.841,E2 -3752.841} C_VEL
LIN {X 0,Y 545.021,Z 220.595,A -85,B 0,C 180,E1 -3755.629,E2 -3755.629} C_VEL
LIN {X 0,Y 545.07,Z 220.588,A -85,B 0,C 180,E1 -3758.18,E2 -3758.18} C_VEL
LIN {X 0,Y 545.122,Z 220.581,A -85,B 0,C 180,E1 -3760.415,E2 -3760.415} C_VEL
LIN {X 0,Y 545.072,Z 220.587,A -85,B 0,C 180,E1 -3763.521,E2 -3763.521} C_VEL
LIN {X 0,Y 545.084,Z 220.587,A -85,B 0,C 180,E1 -3765.82,E2 -3765.82} C_VEL
LIN {X 0,Y 545.078,Z 220.584,A -85,B 0,C 180,E1 -3768.849,E2 -3768.849} C_VEL
LIN {X 0,Y 545.092,Z 220.585,A -85,B 0,C 180,E1 -3771.847,E2 -3771.847} C_VEL
LIN {X 0,Y 545.173,Z 220.575,A -85,B 0,C 180,E1 -3774.081,E2 -3774.081} C_VEL
LIN {X 0,Y 545.174,Z 220.575,A -85,B 0,C 180,E1 -3777.044,E2 -3777.044} C_VEL
LIN {X 0,Y 545.193,Z 220.575,A -85,B 0,C 180,E1 -3780,E2 -3780} C_VEL
LIN {X 0,Y 545.159,Z 220.577,A -85,B 0,C 180,E1 -3782.956,E2 -3782.956} C_VEL
LIN {X 0,Y 545.167,Z 220.574,A -85,B 0,C 180,E1 -3785.92,E2 -3785.92} C_VEL
LIN {X 0,Y 545.106,Z 220.584,A -85,B 0,C 180,E1 -3788.9,E2 -3788.9} C_VEL
LIN {X 0,Y 545.11,Z 220.586,A -85,B 0,C 180,E1 -3791.905,E2 -3791.905} C_VEL
LIN {X 0,Y 545.081,Z 220.588,A -85,B 0,C 180,E1 -3794.944,E2 -3794.944} C_VEL
LIN {X 0,Y 545.057,Z 220.588,A -85,B 0,C 180,E1 -3798.027,E2 -3798.027} C_VEL
LIN {X 0,Y 545.097,Z 220.588,A -85,B 0,C 180,E1 -3800.372,E2 -3800.372} C_VEL
LIN {X 0,Y 545.084,Z 220.589,A -85,B 0,C 180,E1 -3803.559,E2 -3803.559} C_VEL
LIN {X 0,Y 545.081,Z 220.587,A -85,B 0,C 180,E1 -3806.001,E2 -3806.001} C_VEL
LIN {X 0,Y 545.049,Z 220.594,A -85,B 0,C 180,E1 -3808.739,E2 -3808.739} C_VEL
LIN {X 0,Y 545.059,Z 220.588,A -85,B 0,C 180,E1 -3811.915,E2 -3811.915} C_VEL
LIN {X 0,Y 545.064,Z 220.589,A -85,B 0,C 180,E1 -3814.565,E2 -3814.565} C_VEL
LIN {X 0,Y 545.067,Z 220.589,A -85,B 0,C 180,E1 -3816.994,E2 -3816.994} C_VEL
LIN {X 0,Y 544.359,Z 220.681,A -85,B 0,C 180,E1 -3817.61,E2 -3817.61} C_VEL
LIN {X 0,Y 541.493,Z 221.035,A -85,B 0,C 180,E1 -3818.611,E2 -3818.611} C_VEL
LIN {X 0,Y 539.106,Z 221.334,A -85,B 0,C 180,E1 -3819.417,E2 -3819.417} C_VEL
LIN {X 0,Y 538.095,Z 221.456,A -85,B 0,C 180,E1 -3820.039,E2 -3820.039} C_VEL
LIN {X 0,Y 538.02,Z 221.466,A -85,B 0,C 180,E1 -3820.249,E2 -3820.249} C_VEL
LIN {X 0,Y 537.984,Z 221.472,A -85,B 0,C 180,E1 -3822.982,E2 -3822.982} C_VEL
LIN {X 0,Y 538.014,Z 221.47,A -85,B 0,C 180,E1 -3825.928,E2 -3825.928} C_VEL
LIN {X 0,Y 538.026,Z 221.467,A -85,B 0,C 180,E1 -3829.222,E2 -3829.222} C_VEL
LIN {X 0,Y 537.996,Z 221.468,A -85,B 0,C 180,E1 -3832.122,E2 -3832.122} C_VEL
LIN {X 0,Y 537.919,Z 221.482,A -85,B 0,C 180,E1 -3834.909,E2 -3834.909} C_VEL
LIN {X 0,Y 537.805,Z 221.498,A -85,B 0,C 180,E1 -3835.811,E2 -3835.811} C_VEL
LIN {X 0,Y 537.752,Z 223.037,A -85,B 0,C 180,E1 -3837.599,E2 -3837.599} C_VEL
LIN {X 0,Y 537.75,Z 225.834,A -85,B 0,C 180,E1 -3840.222,E2 -3840.222} C_VEL
LIN {X 0,Y 537.724,Z 228.571,A -85,B 0,C 180,E1 -3842.777,E2 -3842.777} C_VEL
LIN {X 0,Y 537.667,Z 231.281,A -85,B 0,C 180,E1 -3845.274,E2 -3845.274} C_VEL
LIN {X 0,Y 537.613,Z 234.906,A -85,B 0,C 180,E1 -3848.529,E2 -3848.529} C_VEL
LIN {X 0,Y 537.568,Z 237.638,A -85,B 0,C 180,E1 -3850.923,E2 -3850.923} C_VEL
LIN {X 0,Y 537.576,Z 240.37,A -85,B 0,C 180,E1 -3853.284,E2 -3853.284} C_VEL
LIN {X 0,Y 537.564,Z 243.109,A -85,B 0,C 180,E1 -3855.617,E2 -3855.617} C_VEL
LIN {X 0,Y 537.528,Z 244.447,A -85,B 0,C 180,E1 -3856.761,E2 -3856.761} C_VEL
LIN {X 0,Y 539.217,Z 253.85,A -85,B 0,C 180,E1 -3857.031,E2 -3857.031} C_VEL
LIN {X 0,Y 539.049,Z 266.786,A -85,B 0,C 180,E1 -3857.481,E2 -3857.481} C_VEL
LIN {X 0,Y 538.849,Z 279.151,A -85,B 0,C 180,E1 -3858.076,E2 -3858.076} C_VEL
LIN {X 0,Y 538.593,Z 290.794,A -85,B 0,C 180,E1 -3858.808,E2 -3858.808} C_VEL
LIN {X 0,Y 538.329,Z 301.459,A -85,B 0,C 180,E1 -3859.659,E2 -3859.659} C_VEL
LIN {X 0,Y 538.135,Z 311.045,A -85,B 0,C 180,E1 -3860.604,E2 -3860.604} C_VEL
LIN {X 0,Y 537.955,Z 318.893,A -85,B 0,C 180,E1 -3861.548,E2 -3861.548} C_VEL
LIN {X 0,Y 537.788,Z 326.566,A -85,B 0,C 180,E1 -3862.68,E2 -3862.68} C_VEL
LIN {X 0,Y 537.717,Z 333.592,A -85,B 0,C 180,E1 -3863.998,E2 -3863.998} C_VEL
LIN {X 0,Y 537.54,Z 338.282,A -85,B 0,C 180,E1 -3865.125,E2 -3865.125} C_VEL
LIN {X 0,Y 537.591,Z 341.864,A -85,B 0,C 180,E1 -3866.252,E2 -3866.252} C_VEL
LIN {X 0,Y 537.551,Z 343.719,A -85,B 0,C 180,E1 -3867.002,E2 -3867.002} C_VEL
LIN {X 0,Y 537.489,Z 345.128,A -85,B 0,C 180,E1 -3867.752,E2 -3867.752} C_VEL
LIN {X 0,Y 537.442,Z 346.757,A -85,B 0,C 180,E1 -3869.251,E2 -3869.251} C_VEL
LIN {X 0,Y 537.442,Z 346.996,A -85,B 0,C 180,E1 -3870,E2 -3870} C_VEL
LIN {X 0,Y 537.442,Z 346.814,A -85,B 0,C 180,E1 -3870.749,E2 -3870.749} C_VEL
LIN {X 0,Y 537.489,Z 345.26,A -85,B 0,C 180,E1 -3872.248,E2 -3872.248} C_VEL
LIN {X 0,Y 537.552,Z 343.906,A -85,B 0,C 180,E1 -3872.998,E2 -3872.998} C_VEL
LIN {X 0,Y 537.603,Z 341.064,A -85,B 0,C 180,E1 -3874.123,E2 -3874.123} C_VEL
LIN {X 0,Y 537.587,Z 337.213,A -85,B 0,C 180,E1 -3875.251,E2 -3875.251} C_VEL
LIN {X 0,Y 537.661,Z 332.516,A -85,B 0,C 180,E1 -3876.32,E2 -3876.32} C_VEL
LIN {X 0,Y 537.79,Z 325.974,A -85,B 0,C 180,E1 -3877.509,E2 -3877.509} C_VEL
LIN {X 0,Y 537.968,Z 318.124,A -85,B 0,C 180,E1 -3878.641,E2 -3878.641} C_VEL
LIN {X 0,Y 538.138,Z 310.12,A -85,B 0,C 180,E1 -3879.585,E2 -3879.585} C_VEL
LIN {X 0,Y 538.365,Z 300.344,A -85,B 0,C 180,E1 -3880.531,E2 -3880.531} C_VEL
LIN {X 0,Y 538.58,Z 290.725,A -85,B 0,C 180,E1 -3881.288,E2 -3881.288} C_VEL
LIN {X 0,Y 538.778,Z 280.348,A -85,B 0,C 180,E1 -3881.95,E2 -3881.95} C_VEL
LIN {X 0,Y 539.037,Z 267.791,A -85,B 0,C 180,E1 -3882.566,E2 -3882.566} C_VEL
LIN {X 0,Y 539.197,Z 255.262,A -85,B 0,C 180,E1 -3883.017,E2 -3883.017} C_VEL
LIN {X 0,Y 538.921,Z 251.844,A -85,B 0,C 180,E1 -3883.12,E2 -3883.12} C_VEL
LIN {X 0,Y 537.545,Z 244.404,A -85,B 0,C 180,E1 -3883.347,E2 -3883.347} C_VEL
LIN {X 0,Y 537.556,Z 241.381,A -85,B 0,C 180,E1 -3885.935,E2 -3885.935} C_VEL
LIN {X 0,Y 537.563,Z 238.689,A -85,B 0,C 180,E1 -3888.287,E2 -3888.287} C_VEL
LIN {X 0,Y 537.58,Z 235.926,A -85,B 0,C 180,E1 -3890.67,E2 -3890.67} C_VEL
LIN {X 0,Y 537.596,Z 233.167,A -85,B 0,C 180,E1 -3893.091,E2 -3893.091} C_VEL
LIN {X 0,Y 537.694,Z 230.409,A -85,B 0,C 180,E1 -3895.594,E2 -3895.594} C_VEL
LIN {X 0,Y 537.721,Z 227.76,A -85,B 0,C 180,E1 -3898.068,E2 -3898.068} C_VEL
LIN {X 0,Y 537.749,Z 225.017,A -85,B 0,C 180,E1 -3900.644,E2 -3900.644} C_VEL
LIN {X 0,Y 537.778,Z 222.202,A -85,B 0,C 180,E1 -3903.29,E2 -3903.29} C_VEL
LIN {X 0,Y 537.797,Z 221.499,A -85,B 0,C 180,E1 -3904.189,E2 -3904.189} C_VEL
LIN {X 0,Y 538.025,Z 221.468,A -85,B 0,C 180,E1 -3906.933,E2 -3906.933} C_VEL
LIN {X 0,Y 538.026,Z 221.464,A -85,B 0,C 180,E1 -3909.797,E2 -3909.797} C_VEL
LIN {X 0,Y 537.99,Z 221.469,A -85,B 0,C 180,E1 -3912.789,E2 -3912.789} C_VEL
LIN {X 0,Y 537.996,Z 221.467,A -85,B 0,C 180,E1 -3915.136,E2 -3915.136} C_VEL
LIN {X 0,Y 538.021,Z 221.465,A -85,B 0,C 180,E1 -3918.226,E2 -3918.226} C_VEL
LIN {X 0,Y 538.015,Z 221.469,A -85,B 0,C 180,E1 -3921.169,E2 -3921.169} C_VEL
LIN {X 0,Y 537.998,Z 221.472,A -85,B 0,C 180,E1 -3924.089,E2 -3924.089} C_VEL
LIN {X 0,Y 538.034,Z 221.463,A -85,B 0,C 180,E1 -3926.727,E2 -3926.727} C_VEL
LIN {X 0,Y 538.004,Z 221.471,A -85,B 0,C 180,E1 -3929.561,E2 -3929.561} C_VEL
LIN {X 0,Y 538.027,Z 221.468,A -85,B 0,C 180,E1 -3932.655,E2 -3932.655} C_VEL
LIN {X 0,Y 538.027,Z 221.465,A -85,B 0,C 180,E1 -3935.291,E2 -3935.291} C_VEL
LIN {X 0,Y 538.019,Z 221.469,A -85,B 0,C 180,E1 -3938.042,E2 -3938.042} C_VEL
LIN {X 0,Y 538.084,Z 221.458,A -85,B 0,C 180,E1 -3940.148,E2 -3940.148} C_VEL
LIN {X 0,Y 537.989,Z 221.472,A -85,B 0,C 180,E1 -3943.298,E2 -3943.298} C_VEL
LIN {X 0,Y 538.041,Z 221.462,A -85,B 0,C 180,E1 -3945.63,E2 -3945.63} C_VEL
LIN {X 0,Y 538.081,Z 221.459,A -85,B 0,C 180,E1 -3948.702,E2 -3948.702} C_VEL
LIN {X 0,Y 538.083,Z 221.461,A -85,B 0,C 180,E1 -3951.739,E2 -3951.739} C_VEL
LIN {X 0,Y 538.118,Z 221.453,A -85,B 0,C 180,E1 -3954.003,E2 -3954.003} C_VEL
LIN {X 0,Y 538.128,Z 221.454,A -85,B 0,C 180,E1 -3957.005,E2 -3957.005} C_VEL
LIN {X 0,Y 538.182,Z 221.446,A -85,B 0,C 180,E1 -3960.748,E2 -3960.748} C_VEL
LIN {X 0,Y 538.139,Z 221.451,A -85,B 0,C 180,E1 -3962.994,E2 -3962.994} C_VEL
LIN {X 0,Y 538.123,Z 221.453,A -85,B 0,C 180,E1 -3965.997,E2 -3965.997} C_VEL
LIN {X 0,Y 538.057,Z 221.462,A -85,B 0,C 180,E1 -3968.261,E2 -3968.261} C_VEL
LIN {X 0,Y 538.042,Z 221.462,A -85,B 0,C 180,E1 -3971.573,E2 -3971.573} C_VEL
LIN {X 0,Y 538.051,Z 221.461,A -85,B 0,C 180,E1 -3974.853,E2 -3974.853} C_VEL
LIN {X 0,Y 538.064,Z 221.463,A -85,B 0,C 180,E1 -3977.54,E2 -3977.54} C_VEL
LIN {X 0,Y 538.041,Z 221.467,A -85,B 0,C 180,E1 -3980.651,E2 -3980.651} C_VEL
LIN {X 0,Y 538.009,Z 221.47,A -85,B 0,C 180,E1 -3983.877,E2 -3983.877} C_VEL
LIN {X 0,Y 537.985,Z 221.469,A -85,B 0,C 180,E1 -3986.37,E2 -3986.37} C_VEL
LIN {X 0,Y 537.994,Z 221.471,A -85,B 0,C 180,E1 -3988.926,E2 -3988.926} C_VEL
LIN {X 0,Y 538.014,Z 221.466,A -85,B 0,C 180,E1 -3991.887,E2 -3991.887} C_VEL
LIN {X 0,Y 538.014,Z 221.469,A -85,B 0,C 180,E1 -3994.617,E2 -3994.617} C_VEL
LIN {X 0,Y 538.001,Z 221.468,A -85,B 0,C 180,E1 -3997.169,E2 -3997.169} C_VEL
LIN {X 0,Y 538.002,Z 221.469,A -85,B 0,C 180,E1 -3999.799,E2 -3999.799} C_VEL
LIN {X 0,Y 538,Z 221.473,A -85,B 0,C 180,E1 -4002.984,E2 -4002.984} C_VEL
LIN {X 0,Y 538.021,Z 221.468,A -85,B 0,C 180,E1 -4005.927,E2 -4005.927} C_VEL
LIN {X 0,Y 538.033,Z 221.469,A -85,B 0,C 180,E1 -4008.227,E2 -4008.227} C_VEL
LIN {X 0,Y 538.012,Z 221.472,A -85,B 0,C 180,E1 -4011.169,E2 -4011.169} C_VEL
LIN {X 0,Y 538.035,Z 221.584,A -85,B 0,C 180,E1 -4012.126,E2 -4012.126} C_VEL
LIN {X 0,Y 538.915,Z 226.99,A -85,B 0,C 180,E1 -4014.066,E2 -4014.066} C_VEL
LIN {X 0,Y 538.955,Z 233.507,A -85,B 0,C 180,E1 -4016.277,E2 -4016.277} C_VEL
LIN {X 0,Y 538.754,Z 241.775,A -85,B 0,C 180,E1 -4018.984,E2 -4018.984} C_VEL
LIN {X 0,Y 538.566,Z 251.042,A -85,B 0,C 180,E1 -4021.98,E2 -4021.98} C_VEL
LIN {X 0,Y 538.397,Z 258.986,A -85,B 0,C 180,E1 -4024.484,E2 -4024.484} C_VEL
LIN {X 0,Y 538.228,Z 268.253,A -85,B 0,C 180,E1 -4027.344,E2 -4027.344} C_VEL
LIN {X 0,Y 538.024,Z 278.844,A -85,B 0,C 180,E1 -4030.543,E2 -4030.543} C_VEL
LIN {X 0,Y 537.892,Z 288.112,A -85,B 0,C 180,E1 -4033.295,E2 -4033.295} C_VEL
LIN {X 0,Y 537.772,Z 297.379,A -85,B 0,C 180,E1 -4036.009,E2 -4036.009} C_VEL
LIN {X 0,Y 537.73,Z 299.53,A -85,B 0,C 180,E1 -4036.634,E2 -4036.634} C_VEL
LIN {X 0,Y 539.248,Z 310.354,A -85,B 0,C 180,E1 -4036.912,E2 -4036.912} C_VEL
LIN {X 0,Y 539.066,Z 322.475,A -85,B 0,C 180,E1 -4037.291,E2 -4037.291} C_VEL
LIN {X 0,Y 538.841,Z 333.487,A -85,B 0,C 180,E1 -4037.764,E2 -4037.764} C_VEL
LIN {X 0,Y 538.603,Z 344.817,A -85,B 0,C 180,E1 -4038.394,E2 -4038.394} C_VEL
LIN {X 0,Y 538.411,Z 355.926,A -85,B 0,C 180,E1 -4039.185,E2 -4039.185} C_VEL
LIN {X 0,Y 538.222,Z 365.602,A -85,B 0,C 180,E1 -4040.037,E2 -4040.037} C_VEL
LIN {X 0,Y 538.015,Z 374.413,A -85,B 0,C 180,E1 -4040.982,E2 -4040.982} C_VEL
LIN {X 0,Y 537.829,Z 383.001,A -85,B 0,C 180,E1 -4042.114,E2 -4042.114} C_VEL
LIN {X 0,Y 537.705,Z 389.868,A -85,B 0,C 180,E1 -4043.245,E2 -4043.245} C_VEL
LIN {X 0,Y 537.676,Z 395.366,A -85,B 0,C 180,E1 -4044.374,E2 -4044.374} C_VEL
LIN {X 0,Y 537.557,Z 399.678,A -85,B 0,C 180,E1 -4045.501,E2 -4045.501} C_VEL
LIN {X 0,Y 537.591,Z 401.958,A -85,B 0,C 180,E1 -4046.252,E2 -4046.252} C_VEL
LIN {X 0,Y 537.551,Z 403.808,A -85,B 0,C 180,E1 -4047.002,E2 -4047.002} C_VEL
LIN {X 0,Y 537.49,Z 405.198,A -85,B 0,C 180,E1 -4047.752,E2 -4047.752} C_VEL
LIN {X 0,Y 537.442,Z 406.785,A -85,B 0,C 180,E1 -4049.251,E2 -4049.251} C_VEL
LIN {X 0,Y 537.442,Z 407,A -85,B 0,C 180,E1 -4050,E2 -4050} C_VEL
LIN {X 0,Y 537.451,Z 406.186,A -85,B 0,C 180,E1 -4051.499,E2 -4051.499} C_VEL
LIN {X 0,Y 537.49,Z 405.199,A -85,B 0,C 180,E1 -4052.248,E2 -4052.248} C_VEL
LIN {X 0,Y 537.551,Z 403.81,A -85,B 0,C 180,E1 -4052.998,E2 -4052.998} C_VEL
LIN {X 0,Y 537.603,Z 400.895,A -85,B 0,C 180,E1 -4054.123,E2 -4054.123} C_VEL
LIN {X 0,Y 537.587,Z 396.948,A -85,B 0,C 180,E1 -4055.251,E2 -4055.251} C_VEL
LIN {X 0,Y 537.652,Z 392.087,A -85,B 0,C 180,E1 -4056.334,E2 -4056.334} C_VEL
LIN {X 0,Y 537.791,Z 385.467,A -85,B 0,C 180,E1 -4057.509,E2 -4057.509} C_VEL
LIN {X 0,Y 537.973,Z 377.477,A -85,B 0,C 180,E1 -4058.641,E2 -4058.641} C_VEL
LIN {X 0,Y 538.118,Z 369.334,A -85,B 0,C 180,E1 -4059.586,E2 -4059.586} C_VEL
LIN {X 0,Y 538.337,Z 359.399,A -85,B 0,C 180,E1 -4060.531,E2 -4060.531} C_VEL
LIN {X 0,Y 538.531,Z 349.584,A -85,B 0,C 180,E1 -4061.289,E2 -4061.289} C_VEL
LIN {X 0,Y 538.716,Z 338.585,A -85,B 0,C 180,E1 -4061.972,E2 -4061.972} C_VEL
LIN {X 0,Y 538.991,Z 326.105,A -85,B 0,C 180,E1 -4062.568,E2 -4062.568} C_VEL
LIN {X 0,Y 539.223,Z 313.082,A -85,B 0,C 180,E1 -4063.017,E2 -4063.017} C_VEL
LIN {X 0,Y 538.96,Z 306.927,A -85,B 0,C 180,E1 -4063.179,E2 -4063.179} C_VEL
LIN {X 0,Y 537.731,Z 299.529,A -85,B 0,C 180,E1 -4063.366,E2 -4063.366} C_VEL
LIN {X 0,Y 537.874,Z 289.435,A -85,B 0,C 180,E1 -4066.316,E2 -4066.316} C_VEL
LIN {X 0,Y 537.994,Z 280.167,A -85,B 0,C 180,E1 -4069.062,E2 -4069.062} C_VEL
LIN {X 0,Y 538.129,Z 272.224,A -85,B 0,C 180,E1 -4071.45,E2 -4071.45} C_VEL
LIN {X 0,Y 538.329,Z 262.958,A -85,B 0,C 180,E1 -4074.283,E2 -4074.283} C_VEL
LIN {X 0,Y 538.527,Z 252.843,A -85,B 0,C 180,E1 -4077.448,E2 -4077.448} C_VEL
LIN {X 0,Y 538.726,Z 243.098,A -85,B 0,C 180,E1 -4080.583,E2 -4080.583} C_VEL
LIN {X 0,Y 538.947,Z 234.381,A -85,B 0,C 180,E1 -4083.428,E2 -4083.428} C_VEL
LIN {X 0,Y 539.024,Z 228.324,A -85,B 0,C 180,E1 -4085.466,E2 -4085.466} C_VEL
LIN {X 0,Y 538.355,Z 223.371,A -85,B 0,C 180,E1 -4087.219,E2 -4087.219} C_VEL
LIN {X 0,Y 537.999,Z 221.473,A -85,B 0,C 180,E1 -4088.006,E2 -4088.006} C_VEL
LIN {X 0,Y 538.052,Z 221.464,A -85,B 0,C 180,E1 -4090.776,E2 -4090.776} C_VEL
LIN {X 0,Y 538.007,Z 221.474,A -85,B 0,C 180,E1 -4093.816,E2 -4093.816} C_VEL
LIN {X 0,Y 538.007,Z 221.467,A -85,B 0,C 180,E1 -4096.184,E2 -4096.184} C_VEL
LIN {X 0,Y 537.998,Z 221.468,A -85,B 0,C 180,E1 -4099.26,E2 -4099.26} C_VEL
LIN {X 0,Y 537.988,Z 221.473,A -85,B 0,C 180,E1 -4102.122,E2 -4102.122} C_VEL
LIN {X 0,Y 537.999,Z 221.468,A -85,B 0,C 180,E1 -4104.916,E2 -4104.916} C_VEL
LIN {X 0,Y 538.024,Z 221.469,A -85,B 0,C 180,E1 -4107.617,E2 -4107.617} C_VEL
LIN {X 0,Y 538.004,Z 221.468,A -85,B 0,C 180,E1 -4110.238,E2 -4110.238} C_VEL
LIN {X 0,Y 538.003,Z 221.469,A -85,B 0,C 180,E1 -4112.793,E2 -4112.793} C_VEL
LIN {X 0,Y 537.983,Z 221.469,A -85,B 0,C 180,E1 -4115.289,E2 -4115.289} C_VEL
LIN {X 0,Y 538.02,Z 221.467,A -85,B 0,C 180,E1 -4118.042,E2 -4118.042} C_VEL
LIN {X 0,Y 538.039,Z 221.467,A -85,B 0,C 180,E1 -4120.94,E2 -4120.94} C_VEL
LIN {X 0,Y 538.021,Z 221.466,A -85,B 0,C 180,E1 -4123.299,E2 -4123.299} C_VEL
LIN {X 0,Y 538.054,Z 221.461,A -85,B 0,C 180,E1 -4125.63,E2 -4125.63} C_VEL
LIN {X 0,Y 538.031,Z 221.462,A -85,B 0,C 180,E1 -4128.701,E2 -4128.701} C_VEL
LIN {X 0,Y 538.057,Z 221.462,A -85,B 0,C 180,E1 -4131.739,E2 -4131.739} C_VEL
LIN {X 0,Y 538.124,Z 221.452,A -85,B 0,C 180,E1 -4134.003,E2 -4134.003} C_VEL
LIN {X 0,Y 538.141,Z 221.451,A -85,B 0,C 180,E1 -4137.006,E2 -4137.006} C_VEL
LIN {X 0,Y 538.162,Z 221.451,A -85,B 0,C 180,E1 -4140,E2 -4140} C_VEL
LIN {X 0,Y 538.127,Z 221.453,A -85,B 0,C 180,E1 -4142.995,E2 -4142.995} C_VEL
LIN {X 0,Y 538.119,Z 221.453,A -85,B 0,C 180,E1 -4145.997,E2 -4145.997} C_VEL
LIN {X 0,Y 538.065,Z 221.463,A -85,B 0,C 180,E1 -4148.261,E2 -4148.261} C_VEL
LIN {X 0,Y 538.092,Z 221.46,A -85,B 0,C 180,E1 -4151.598,E2 -4151.598} C_VEL
LIN {X 0,Y 538.048,Z 221.463,A -85,B 0,C 180,E1 -4154.85,E2 -4154.85} C_VEL
LIN {X 0,Y 538.012,Z 221.467,A -85,B 0,C 180,E1 -4158.271,E2 -4158.271} C_VEL
LIN {X 0,Y 538.042,Z 221.466,A -85,B 0,C 180,E1 -4160.651,E2 -4160.651} C_VEL
LIN {X 0,Y 538.008,Z 221.471,A -85,B 0,C 180,E1 -4163.888,E2 -4163.888} C_VEL
LIN {X 0,Y 538.041,Z 221.463,A -85,B 0,C 180,E1 -4166.367,E2 -4166.367} C_VEL
LIN {X 0,Y 537.996,Z 221.473,A -85,B 0,C 180,E1 -4168.926,E2 -4168.926} C_VEL
LIN {X 0,Y 538.014,Z 221.466,A -85,B 0,C 180,E1 -4171.887,E2 -4171.887} C_VEL
LIN {X 0,Y 538.014,Z 221.467,A -85,B 0,C 180,E1 -4174.617,E2 -4174.617} C_VEL
LIN {X 0,Y 538.009,Z 221.47,A -85,B 0,C 180,E1 -4177.17,E2 -4177.17} C_VEL
LIN {X 0,Y 538.02,Z 221.466,A -85,B 0,C 180,E1 -4180.249,E2 -4180.249} C_VEL
LIN {X 0,Y 537.367,Z 221.551,A -85,B 0,C 180,E1 -4180.875,E2 -4180.875} C_VEL
LIN {X 0,Y 534.506,Z 221.906,A -85,B 0,C 180,E1 -4181.889,E2 -4181.889} C_VEL
LIN {X 0,Y 532.075,Z 222.209,A -85,B 0,C 180,E1 -4182.706,E2 -4182.706} C_VEL
LIN {X 0,Y 531.026,Z 222.336,A -85,B 0,C 180,E1 -4183.337,E2 -4183.337} C_VEL
LIN {X 0,Y 530.939,Z 222.346,A -85,B 0,C 180,E1 -4183.551,E2 -4183.551} C_VEL
LIN {X 0,Y 530.941,Z 222.347,A -85,B 0,C 180,E1 -4186.502,E2 -4186.502} C_VEL
LIN {X 0,Y 530.965,Z 222.345,A -85,B 0,C 180,E1 -4188.979,E2 -4188.979} C_VEL
LIN {X 0,Y 530.961,Z 222.347,A -85,B 0,C 180,E1 -4191.529,E2 -4191.529} C_VEL
LIN {X 0,Y 530.905,Z 222.356,A -85,B 0,C 180,E1 -4194.376,E2 -4194.376} C_VEL
LIN {X 0,Y 530.71,Z 222.381,A -85,B 0,C 180,E1 -4196.207,E2 -4196.207} C_VEL
LIN {X 0,Y 530.693,Z 225.635,A -85,B 0,C 180,E1 -4199.407,E2 -4199.407} C_VEL
LIN {X 0,Y 530.66,Z 228.966,A -85,B 0,C 180,E1 -4202.541,E2 -4202.541} C_VEL
LIN {X 0,Y 530.596,Z 231.517,A -85,B 0,C 180,E1 -4204.921,E2 -4204.921} C_VEL
LIN {X 0,Y 530.547,Z 234.912,A -85,B 0,C 180,E1 -4208.014,E2 -4208.014} C_VEL
LIN {X 0,Y 530.517,Z 237.903,A -85,B 0,C 180,E1 -4210.659,E2 -4210.659} C_VEL
LIN {X 0,Y 530.507,Z 240.672,A -85,B 0,C 180,E1 -4213.055,E2 -4213.055} C_VEL
LIN {X 0,Y 530.525,Z 243.534,A -85,B 0,C 180,E1 -4215.422,E2 -4215.422} C_VEL
LIN {X 0,Y 530.486,Z 244.912,A -85,B 0,C 180,E1 -4216.582,E2 -4216.582} C_VEL
LIN {X 0,Y 532.307,Z 255.117,A -85,B 0,C 180,E1 -4216.884,E2 -4216.884} C_VEL
LIN {X 0,Y 532.132,Z 268.35,A -85,B 0,C 180,E1 -4217.364,E2 -4217.364} C_VEL
LIN {X 0,Y 531.924,Z 279.867,A -85,B 0,C 180,E1 -4217.934,E2 -4217.934} C_VEL
LIN {X 0,Y 531.634,Z 291.23,A -85,B 0,C 180,E1 -4218.659,E2 -4218.659} C_VEL
LIN {X 0,Y 531.367,Z 301.892,A -85,B 0,C 180,E1 -4219.522,E2 -4219.522} C_VEL
LIN {X 0,Y 531.153,Z 311.476,A -85,B 0,C 180,E1 -4220.48,E2 -4220.48} C_VEL
LIN {X 0,Y 530.938,Z 319.325,A -85,B 0,C 180,E1 -4221.436,E2 -4221.436} C_VEL
LIN {X 0,Y 530.764,Z 326.996,A -85,B 0,C 180,E1 -4222.582,E2 -4222.582} C_VEL
LIN {X 0,Y 530.652,Z 334.022,A -85,B 0,C 180,E1 -4223.918,E2 -4223.918} C_VEL
LIN {X 0,Y 530.486,Z 338.711,A -85,B 0,C 180,E1 -4225.06,E2 -4225.06} C_VEL
LIN {X 0,Y 530.516,Z 342.292,A -85,B 0,C 180,E1 -4226.202,E2 -4226.202} C_VEL
LIN {X 0,Y 530.486,Z 344.146,A -85,B 0,C 180,E1 -4226.962,E2 -4226.962} C_VEL
LIN {X 0,Y 530.41,Z 345.549,A -85,B 0,C 180,E1 -4227.722,E2 -4227.722} C_VEL
LIN {X 0,Y 530.354,Z 347.159,A -85,B 0,C 180,E1 -4229.241,E2 -4229.241} C_VEL
LIN {X 0,Y 530.354,Z 347.395,A -85,B 0,C 180,E1 -4230,E2 -4230} C_VEL
LIN {X 0,Y 530.354,Z 347.214,A -85,B 0,C 180,E1 -4230.759,E2 -4230.759} C_VEL
LIN {X 0,Y 530.41,Z 345.678,A -85,B 0,C 180,E1 -4232.278,E2 -4232.278} C_VEL
LIN {X 0,Y 530.487,Z 344.331,A -85,B 0,C 180,E1 -4233.038,E2 -4233.038} C_VEL
LIN {X 0,Y 530.523,Z 341.49,A -85,B 0,C 180,E1 -4234.178,E2 -4234.178} C_VEL
LIN {X 0,Y 530.525,Z 337.638,A -85,B 0,C 180,E1 -4235.321,E2 -4235.321} C_VEL
LIN {X 0,Y 530.633,Z 331.919,A -85,B 0,C 180,E1 -4236.613,E2 -4236.613} C_VEL
LIN {X 0,Y 530.792,Z 325.181,A -85,B 0,C 180,E1 -4237.8,E2 -4237.8} C_VEL
LIN {X 0,Y 530.971,Z 317.076,A -85,B 0,C 180,E1 -4238.947,E2 -4238.947} C_VEL
LIN {X 0,Y 531.2,Z 308.775,A -85,B 0,C 180,E1 -4239.904,E2 -4239.904} C_VEL
LIN {X 0,Y 531.455,Z 298.522,A -85,B 0,C 180,E1 -4240.862,E2 -4240.862} C_VEL
LIN {X 0,Y 531.742,Z 287.774,A -85,B 0,C 180,E1 -4241.668,E2 -4241.668} C_VEL
LIN {X 0,Y 531.982,Z 277.232,A -85,B 0,C 180,E1 -4242.3,E2 -4242.3} C_VEL
LIN {X 0,Y 532.194,Z 264.738,A -85,B 0,C 180,E1 -4242.876,E2 -4242.876} C_VEL
LIN {X 0,Y 532.272,Z 254.058,A -85,B 0,C 180,E1 -4243.238,E2 -4243.238} C_VEL
LIN {X 0,Y 530.465,Z 244.794,A -85,B 0,C 180,E1 -4243.528,E2 -4243.528} C_VEL
LIN {X 0,Y 530.504,Z 241.71,A -85,B 0,C 180,E1 -4246.153,E2 -4246.153} C_VEL
LIN {X 0,Y 530.485,Z 238.945,A -85,B 0,C 180,E1 -4248.539,E2 -4248.539} C_VEL
LIN {X 0,Y 530.53,Z 236.174,A -85,B 0,C 180,E1 -4250.957,E2 -4250.957} C_VEL
LIN {X 0,Y 530.565,Z 232.486,A -85,B 0,C 180,E1 -4254.245,E2 -4254.245} C_VEL
LIN {X 0,Y 530.616,Z 229.793,A -85,B 0,C 180,E1 -4256.765,E2 -4256.765} C_VEL
LIN {X 0,Y 530.665,Z 227.063,A -85,B 0,C 180,E1 -4259.342,E2 -4259.342} C_VEL
LIN {X 0,Y 530.675,Z 224.198,A -85,B 0,C 180,E1 -4262.05,E2 -4262.05} C_VEL
LIN {X 0,Y 530.706,Z 222.382,A -85,B 0,C 180,E1 -4263.793,E2 -4263.793} C_VEL
LIN {X 0,Y 530.943,Z 222.348,A -85,B 0,C 180,E1 -4266.56,E2 -4266.56} C_VEL
LIN {X 0,Y 530.99,Z 222.342,A -85,B 0,C 180,E1 -4269.443,E2 -4269.443} C_VEL
LIN {X 0,Y 530.961,Z 222.348,A -85,B 0,C 180,E1 -4272.459,E2 -4272.459} C_VEL
LIN {X 0,Y 530.972,Z 222.347,A -85,B 0,C 180,E1 -4275.623,E2 -4275.623} C_VEL
LIN {X 0,Y 530.982,Z 222.343,A -85,B 0,C 180,E1 -4278.563,E2 -4278.563} C_VEL
LIN {X 0,Y 530.959,Z 222.346,A -85,B 0,C 180,E1 -4281.529,E2 -4281.529} C_VEL
LIN {X 0,Y 530.957,Z 222.349,A -85,B 0,C 180,E1 -4284.38,E2 -4284.38} C_VEL
LIN {X 0,Y 530.969,Z 222.343,A -85,B 0,C 180,E1 -4287.133,E2 -4287.133} C_VEL
LIN {X 0,Y 530.949,Z 222.347,A -85,B 0,C 180,E1 -4289.802,E2 -4289.802} C_VEL
LIN {X 0,Y 530.973,Z 222.345,A -85,B 0,C 180,E1 -4292.477,E2 -4292.477} C_VEL
LIN {X 0,Y 530.992,Z 222.343,A -85,B 0,C 180,E1 -4294.942,E2 -4294.942} C_VEL
LIN {X 0,Y 530.975,Z 222.346,A -85,B 0,C 180,E1 -4298.247,E2 -4298.247} C_VEL
LIN {X 0,Y 530.985,Z 222.341,A -85,B 0,C 180,E1 -4300.677,E2 -4300.677} C_VEL
LIN {X 0,Y 530.956,Z 222.351,A -85,B 0,C 180,E1 -4303.07,E2 -4303.07} C_VEL
LIN {X 0,Y 531.002,Z 222.339,A -85,B 0,C 180,E1 -4305.435,E2 -4305.435} C_VEL
LIN {X 0,Y 531.039,Z 222.338,A -85,B 0,C 180,E1 -4308.55,E2 -4308.55} C_VEL
LIN {X 0,Y 531.054,Z 222.337,A -85,B 0,C 180,E1 -4311.629,E2 -4311.629} C_VEL
LIN {X 0,Y 531.116,Z 222.327,A -85,B 0,C 180,E1 -4314.685,E2 -4314.685} C_VEL
LIN {X 0,Y 531.128,Z 222.322,A -85,B 0,C 180,E1 -4317.725,E2 -4317.725} C_VEL
LIN {X 0,Y 531.152,Z 222.321,A -85,B 0,C 180,E1 -4320.758,E2 -4320.758} C_VEL
LIN {X 0,Y 531.106,Z 222.328,A -85,B 0,C 180,E1 -4323.034,E2 -4323.034} C_VEL
LIN {X 0,Y 531.079,Z 222.33,A -85,B 0,C 180,E1 -4326.077,E2 -4326.077} C_VEL
LIN {X 0,Y 531.011,Z 222.339,A -85,B 0,C 180,E1 -4329.138,E2 -4329.138} C_VEL
LIN {X 0,Y 531.009,Z 222.343,A -85,B 0,C 180,E1 -4332.226,E2 -4332.226} C_VEL
LIN {X 0,Y 530.996,Z 222.343,A -85,B 0,C 180,E1 -4335.35,E2 -4335.35} C_VEL
LIN {X 0,Y 530.992,Z 222.343,A -85,B 0,C 180,E1 -4338.521,E2 -4338.521} C_VEL
LIN {X 0,Y 531.003,Z 222.343,A -85,B 0,C 180,E1 -4340.938,E2 -4340.938} C_VEL
LIN {X 0,Y 530.951,Z 222.349,A -85,B 0,C 180,E1 -4344.226,E2 -4344.226} C_VEL
LIN {X 0,Y 530.95,Z 222.344,A -85,B 0,C 180,E1 -4346.747,E2 -4346.747} C_VEL
LIN {X 0,Y 530.964,Z 222.35,A -85,B 0,C 180,E1 -4349.324,E2 -4349.324} C_VEL
LIN {X 0,Y 530.969,Z 222.345,A -85,B 0,C 180,E1 -4352.1,E2 -4352.1} C_VEL
LIN {X 0,Y 530.971,Z 222.345,A -85,B 0,C 180,E1 -4354.851,E2 -4354.851} C_VEL
LIN {X 0,Y 530.965,Z 222.348,A -85,B 0,C 180,E1 -4357.508,E2 -4357.508} C_VEL
LIN {X 0,Y 530.944,Z 222.345,A -85,B 0,C 180,E1 -4360.437,E2 -4360.437} C_VEL
LIN {X 0,Y 530.947,Z 222.347,A -85,B 0,C 180,E1 -4363.497,E2 -4363.497} C_VEL
LIN {X 0,Y 530.957,Z 222.349,A -85,B 0,C 180,E1 -4366.504,E2 -4366.504} C_VEL
LIN {X 0,Y 530.986,Z 222.343,A -85,B 0,C 180,E1 -4368.976,E2 -4368.976} C_VEL
LIN {X 0,Y 530.987,Z 222.457,A -85,B 0,C 180,E1 -4371.894,E2 -4371.894} C_VEL
LIN {X 0,Y 531.978,Z 228.463,A -85,B 0,C 180,E1 -4374.089,E2 -4374.089} C_VEL
LIN {X 0,Y 531.981,Z 234.992,A -85,B 0,C 180,E1 -4376.335,E2 -4376.335} C_VEL
LIN {X 0,Y 531.756,Z 243.766,A -85,B 0,C 180,E1 -4379.214,E2 -4379.214} C_VEL
LIN {X 0,Y 531.526,Z 253.69,A -85,B 0,C 180,E1 -4382.433,E2 -4382.433} C_VEL
LIN {X 0,Y 531.332,Z 262.957,A -85,B 0,C 180,E1 -4385.376,E2 -4385.376} C_VEL
LIN {X 0,Y 531.118,Z 272.225,A -85,B 0,C 180,E1 -4388.253,E2 -4388.253} C_VEL
LIN {X 0,Y 530.958,Z 281.492,A -85,B 0,C 180,E1 -4391.077,E2 -4391.077} C_VEL
LIN {X 0,Y 530.813,Z 290.759,A -85,B 0,C 180,E1 -4393.857,E2 -4393.857} C_VEL
LIN {X 0,Y 530.689,Z 299.53,A -85,B 0,C 180,E1 -4396.453,E2 -4396.453} C_VEL
LIN {X 0,Y 532.346,Z 310.353,A -85,B 0,C 180,E1 -4396.739,E2 -4396.739} C_VEL
LIN {X 0,Y 532.129,Z 323.77,A -85,B 0,C 180,E1 -4397.171,E2 -4397.171} C_VEL
LIN {X 0,Y 531.86,Z 335.411,A -85,B 0,C 180,E1 -4397.697,E2 -4397.697} C_VEL
LIN {X 0,Y 531.625,Z 346.563,A -85,B 0,C 180,E1 -4398.356,E2 -4398.356} C_VEL
LIN {X 0,Y 531.351,Z 358.261,A -85,B 0,C 180,E1 -4399.232,E2 -4399.232} C_VEL
LIN {X 0,Y 531.118,Z 367.539,A -85,B 0,C 180,E1 -4400.095,E2 -4400.095} C_VEL
LIN {X 0,Y 530.931,Z 375.991,A -85,B 0,C 180,E1 -4401.052,E2 -4401.052} C_VEL
LIN {X 0,Y 530.758,Z 384.238,A -85,B 0,C 180,E1 -4402.2,E2 -4402.2} C_VEL
LIN {X 0,Y 530.598,Z 391.27,A -85,B 0,C 180,E1 -4403.419,E2 -4403.419} C_VEL
LIN {X 0,Y 530.524,Z 396.95,A -85,B 0,C 180,E1 -4404.679,E2 -4404.679} C_VEL
LIN {X 0,Y 530.522,Z 400.895,A -85,B 0,C 180,E1 -4405.822,E2 -4405.822} C_VEL
LIN {X 0,Y 530.457,Z 403.808,A -85,B 0,C 180,E1 -4406.962,E2 -4406.962} C_VEL
LIN {X 0,Y 530.411,Z 405.198,A -85,B 0,C 180,E1 -4407.722,E2 -4407.722} C_VEL
LIN {X 0,Y 530.344,Z 406.785,A -85,B 0,C 180,E1 -4409.241,E2 -4409.241} C_VEL
LIN {X 0,Y 530.342,Z 407,A -85,B 0,C 180,E1 -4410,E2 -4410} C_VEL
LIN {X 0,Y 530.361,Z 406.186,A -85,B 0,C 180,E1 -4411.519,E2 -4411.519} C_VEL
LIN {X 0,Y 530.411,Z 405.199,A -85,B 0,C 180,E1 -4412.278,E2 -4412.278} C_VEL
LIN {X 0,Y 530.457,Z 403.81,A -85,B 0,C 180,E1 -4413.038,E2 -4413.038} C_VEL
LIN {X 0,Y 530.523,Z 400.895,A -85,B 0,C 180,E1 -4414.178,E2 -4414.178} C_VEL
LIN {X 0,Y 530.524,Z 396.948,A -85,B 0,C 180,E1 -4415.321,E2 -4415.321} C_VEL
LIN {X 0,Y 530.6,Z 391.26,A -85,B 0,C 180,E1 -4416.583,E2 -4416.583} C_VEL
LIN {X 0,Y 530.758,Z 384.236,A -85,B 0,C 180,E1 -4417.801,E2 -4417.801} C_VEL
LIN {X 0,Y 530.931,Z 375.989,A -85,B 0,C 180,E1 -4418.948,E2 -4418.948} C_VEL
LIN {X 0,Y 531.118,Z 367.537,A -85,B 0,C 180,E1 -4419.906,E2 -4419.906} C_VEL
LIN {X 0,Y 531.393,Z 357.095,A -85,B 0,C 180,E1 -4420.863,E2 -4420.863} C_VEL
LIN {X 0,Y 531.635,Z 346.444,A -85,B 0,C 180,E1 -4421.651,E2 -4421.651} C_VEL
LIN {X 0,Y 531.86,Z 335.406,A -85,B 0,C 180,E1 -4422.303,E2 -4422.303} C_VEL
LIN {X 0,Y 532.129,Z 323.758,A -85,B 0,C 180,E1 -4422.83,E2 -4422.83} C_VEL
LIN {X 0,Y 532.319,Z 310.34,A -85,B 0,C 180,E1 -4423.262,E2 -4423.262} C_VEL
LIN {X 0,Y 530.689,Z 299.529,A -85,B 0,C 180,E1 -4423.547,E2 -4423.547} C_VEL
LIN {X 0,Y 530.813,Z 290.759,A -85,B 0,C 180,E1 -4426.144,E2 -4426.144} C_VEL
LIN {X 0,Y 530.956,Z 281.491,A -85,B 0,C 180,E1 -4428.923,E2 -4428.923} C_VEL
LIN {X 0,Y 531.118,Z 272.224,A -85,B 0,C 180,E1 -4431.747,E2 -4431.747} C_VEL
LIN {X 0,Y 531.333,Z 262.957,A -85,B 0,C 180,E1 -4434.624,E2 -4434.624} C_VEL
LIN {X 0,Y 531.539,Z 253.459,A -85,B 0,C 180,E1 -4437.641,E2 -4437.641} C_VEL
LIN {X 0,Y 531.756,Z 243.766,A -85,B 0,C 180,E1 -4440.787,E2 -4440.787} C_VEL
LIN {X 0,Y 531.983,Z 234.87,A -85,B 0,C 180,E1 -4443.701,E2 -4443.701} C_VEL
LIN {X 0,Y 531.991,Z 228.433,A -85,B 0,C 180,E1 -4445.909,E2 -4445.909} C_VEL
LIN {X 0,Y 530.975,Z 222.349,A -85,B 0,C 180,E1 -4448.228,E2 -4448.228} C_VEL
LIN {X 0,Y 530.997,Z 222.343,A -85,B 0,C 180,E1 -4451.436,E2 -4451.436} C_VEL
LIN {X 0,Y 530.977,Z 222.344,A -85,B 0,C 180,E1 -4454.549,E2 -4454.549} C_VEL
LIN {X 0,Y 530.941,Z 222.348,A -85,B 0,C 180,E1 -4457.539,E2 -4457.539} C_VEL
LIN {X 0,Y 530.967,Z 222.349,A -85,B 0,C 180,E1 -4460.555,E2 -4460.555} C_VEL
LIN {X 0,Y 530.954,Z 222.346,A -85,B 0,C 180,E1 -4463.441,E2 -4463.441} C_VEL
LIN {X 0,Y 531.003,Z 222.34,A -85,B 0,C 180,E1 -4466.494,E2 -4466.494} C_VEL
LIN {X 0,Y 530.966,Z 222.347,A -85,B 0,C 180,E1 -4469.357,E2 -4469.357} C_VEL
LIN {X 0,Y 530.963,Z 222.35,A -85,B 0,C 180,E1 -4472.479,E2 -4472.479} C_VEL
LIN {X 0,Y 530.95,Z 222.345,A -85,B 0,C 180,E1 -4474.94,E2 -4474.94} C_VEL
LIN {X 0,Y 530.982,Z 222.346,A -85,B 0,C 180,E1 -4477.898,E2 -4477.898} C_VEL
LIN {X 0,Y 530.998,Z 222.342,A -85,B 0,C 180,E1 -4480.677,E2 -4480.677} C_VEL
LIN {X 0,Y 530.978,Z 222.346,A -85,B 0,C 180,E1 -4483.071,E2 -4483.071} C_VEL
LIN {X 0,Y 531.012,Z 222.338,A -85,B 0,C 180,E1 -4485.436,E2 -4485.436} C_VEL
LIN {X 0,Y 530.993,Z 222.339,A -85,B 0,C 180,E1 -4488.549,E2 -4488.549} C_VEL
LIN {X 0,Y 531.033,Z 222.338,A -85,B 0,C 180,E1 -4491.629,E2 -4491.629} C_VEL
LIN {X 0,Y 531.08,Z 222.33,A -85,B 0,C 180,E1 -4493.923,E2 -4493.923} C_VEL
LIN {X 0,Y 531.108,Z 222.328,A -85,B 0,C 180,E1 -4496.966,E2 -4496.966} C_VEL
LIN {X 0,Y 531.131,Z 222.327,A -85,B 0,C 180,E1 -4500,E2 -4500} C_VEL
LIN {X 0,Y 531.095,Z 222.33,A -85,B 0,C 180,E1 -4503.034,E2 -4503.034} C_VEL
LIN {X 0,Y 531.075,Z 222.33,A -85,B 0,C 180,E1 -4506.077,E2 -4506.077} C_VEL
LIN {X 0,Y 531.021,Z 222.338,A -85,B 0,C 180,E1 -4509.138,E2 -4509.138} C_VEL
LIN {X 0,Y 531.055,Z 222.338,A -85,B 0,C 180,E1 -4511.671,E2 -4511.671} C_VEL
LIN {X 0,Y 531.024,Z 222.339,A -85,B 0,C 180,E1 -4514.95,E2 -4514.95} C_VEL
LIN {X 0,Y 530.977,Z 222.341,A -85,B 0,C 180,E1 -4517.724,E2 -4517.724} C_VEL
LIN {X 0,Y 531.03,Z 222.338,A -85,B 0,C 180,E1 -4520.127,E2 -4520.127} C_VEL
LIN {X 0,Y 530.951,Z 222.348,A -85,B 0,C 180,E1 -4522.573,E2 -4522.573} C_VEL
LIN {X 0,Y 530.994,Z 222.342,A -85,B 0,C 180,E1 -4525.058,E2 -4525.058} C_VEL
LIN {X 0,Y 530.969,Z 222.346,A -85,B 0,C 180,E1 -4527.598,E2 -4527.598} C_VEL
LIN {X 0,Y 530.956,Z 222.351,A -85,B 0,C 180,E1 -4530.641,E2 -4530.641} C_VEL
LIN {X 0,Y 530.967,Z 222.344,A -85,B 0,C 180,E1 -4533.5,E2 -4533.5} C_VEL
LIN {X 0,Y 530.949,Z 222.348,A -85,B 0,C 180,E1 -4536.153,E2 -4536.153} C_VEL
LIN {X 0,Y 530.969,Z 222.345,A -85,B 0,C 180,E1 -4538.653,E2 -4538.653} C_VEL
LIN {X 0,Y 530.99,Z 222.342,A -85,B 0,C 180,E1 -4541.436,E2 -4541.436} C_VEL
LIN {X 0,Y 530.939,Z 222.346,A -85,B 0,C 180,E1 -4543.551,E2 -4543.551} C_VEL
LIN {X 0,Y 530.269,Z 222.435,A -85,B 0,C 180,E1 -4544.184,E2 -4544.184} C_VEL
LIN {X 0,Y 527.417,Z 222.785,A -85,B 0,C 180,E1 -4545.213,E2 -4545.213} C_VEL
LIN {X 0,Y 525.01,Z 223.092,A -85,B 0,C 180,E1 -4546.042,E2 -4546.042} C_VEL
LIN {X 0,Y 523.978,Z 223.214,A -85,B 0,C 180,E1 -4546.681,E2 -4546.681} C_VEL
LIN {X 0,Y 523.894,Z 223.223,A -85,B 0,C 180,E1 -4546.898,E2 -4546.898} C_VEL
LIN {X 0,Y 523.953,Z 223.219,A -85,B 0,C 180,E1 -4549.92,E2 -4549.92} C_VEL
LIN {X 0,Y 523.907,Z 223.227,A -85,B 0,C 180,E1 -4552.867,E2 -4552.867} C_VEL
LIN {X 0,Y 523.739,Z 223.25,A -85,B 0,C 180,E1 -4555.695,E2 -4555.695} C_VEL
LIN {X 0,Y 523.668,Z 223.412,A -85,B 0,C 180,E1 -4556.615,E2 -4556.615} C_VEL
LIN {X 0,Y 523.648,Z 226.251,A -85,B 0,C 180,E1 -4559.335,E2 -4559.335} C_VEL
LIN {X 0,Y 523.606,Z 229.426,A -85,B 0,C 180,E1 -4562.36,E2 -4562.36} C_VEL
LIN {X 0,Y 523.514,Z 232.678,A -85,B 0,C 180,E1 -4565.407,E2 -4565.407} C_VEL
LIN {X 0,Y 523.463,Z 235.397,A -85,B 0,C 180,E1 -4567.918,E2 -4567.918} C_VEL
LIN {X 0,Y 523.436,Z 238.148,A -85,B 0,C 180,E1 -4570.387,E2 -4570.387} C_VEL
LIN {X 0,Y 523.424,Z 240.974,A -85,B 0,C 180,E1 -4572.819,E2 -4572.819} C_VEL
LIN {X 0,Y 523.427,Z 244.874,A -85,B 0,C 180,E1 -4576.014,E2 -4576.014} C_VEL
LIN {X 0,Y 523.426,Z 245.379,A -85,B 0,C 180,E1 -4576.398,E2 -4576.398} C_VEL
LIN {X 0,Y 525.43,Z 255.561,A -85,B 0,C 180,E1 -4576.709,E2 -4576.709} C_VEL
LIN {X 0,Y 525.244,Z 268.79,A -85,B 0,C 180,E1 -4577.196,E2 -4577.196} C_VEL
LIN {X 0,Y 525.001,Z 279.888,A -85,B 0,C 180,E1 -4577.749,E2 -4577.749} C_VEL
LIN {X 0,Y 524.694,Z 291.664,A -85,B 0,C 180,E1 -4578.507,E2 -4578.507} C_VEL
LIN {X 0,Y 524.405,Z 302.325,A -85,B 0,C 180,E1 -4579.381,E2 -4579.381} C_VEL
LIN {X 0,Y 524.176,Z 311.908,A -85,B 0,C 180,E1 -4580.352,E2 -4580.352} C_VEL
LIN {X 0,Y 523.933,Z 319.756,A -85,B 0,C 180,E1 -4581.32,E2 -4581.32} C_VEL
LIN {X 0,Y 523.722,Z 327.427,A -85,B 0,C 180,E1 -4582.482,E2 -4582.482} C_VEL
LIN {X 0,Y 523.596,Z 334.453,A -85,B 0,C 180,E1 -4583.836,E2 -4583.836} C_VEL
LIN {X 0,Y 523.432,Z 339.14,A -85,B 0,C 180,E1 -4584.993,E2 -4584.993} C_VEL
LIN {X 0,Y 523.443,Z 342.721,A -85,B 0,C 180,E1 -4586.151,E2 -4586.151} C_VEL
LIN {X 0,Y 523.423,Z 344.574,A -85,B 0,C 180,E1 -4586.921,E2 -4586.921} C_VEL
LIN {X 0,Y 523.335,Z 345.977,A -85,B 0,C 180,E1 -4587.691,E2 -4587.691} C_VEL
LIN {X 0,Y 523.268,Z 347.586,A -85,B 0,C 180,E1 -4589.23,E2 -4589.23} C_VEL
LIN {X 0,Y 523.268,Z 347.822,A -85,B 0,C 180,E1 -4590,E2 -4590} C_VEL
LIN {X 0,Y 523.268,Z 347.641,A -85,B 0,C 180,E1 -4590.769,E2 -4590.769} C_VEL
LIN {X 0,Y 523.335,Z 346.103,A -85,B 0,C 180,E1 -4592.309,E2 -4592.309} C_VEL
LIN {X 0,Y 523.424,Z 344.756,A -85,B 0,C 180,E1 -4593.079,E2 -4593.079} C_VEL
LIN {X 0,Y 523.45,Z 341.915,A -85,B 0,C 180,E1 -4594.235,E2 -4594.235} C_VEL
LIN {X 0,Y 523.464,Z 338.063,A -85,B 0,C 180,E1 -4595.393,E2 -4595.393} C_VEL
LIN {X 0,Y 523.594,Z 332.625,A -85,B 0,C 180,E1 -4596.647,E2 -4596.647} C_VEL
LIN {X 0,Y 523.78,Z 325.603,A -85,B 0,C 180,E1 -4597.905,E2 -4597.905} C_VEL
LIN {X 0,Y 523.971,Z 317.499,A -85,B 0,C 180,E1 -4599.068,E2 -4599.068} C_VEL
LIN {X 0,Y 524.235,Z 309.195,A -85,B 0,C 180,E1 -4600.037,E2 -4600.037} C_VEL
LIN {X 0,Y 524.498,Z 298.941,A -85,B 0,C 180,E1 -4601.008,E2 -4601.008} C_VEL
LIN {X 0,Y 524.814,Z 288.419,A -85,B 0,C 180,E1 -4601.808,E2 -4601.808} C_VEL
LIN {X 0,Y 525.069,Z 277.647,A -85,B 0,C 180,E1 -4602.464,E2 -4602.464} C_VEL
LIN {X 0,Y 525.295,Z 265.148,A -85,B 0,C 180,E1 -4603.048,E2 -4603.048} C_VEL
LIN {X 0,Y 525.233,Z 254.47,A -85,B 0,C 180,E1 -4603.419,E2 -4603.419} C_VEL
LIN {X 0,Y 523.387,Z 245.183,A -85,B 0,C 180,E1 -4603.715,E2 -4603.715} C_VEL
LIN {X 0,Y 523.429,Z 242.035,A -85,B 0,C 180,E1 -4606.377,E2 -4606.377} C_VEL
LIN {X 0,Y 523.426,Z 239.211,A -85,B 0,C 180,E1 -4608.799,E2 -4608.799} C_VEL
LIN {X 0,Y 523.449,Z 236.401,A -85,B 0,C 180,E1 -4611.254,E2 -4611.254} C_VEL
LIN {X 0,Y 523.497,Z 233.268,A -85,B 0,C 180,E1 -4614.089,E2 -4614.089} C_VEL
LIN {X 0,Y 523.544,Z 230.935,A -85,B 0,C 180,E1 -4616.295,E2 -4616.295} C_VEL
LIN {X 0,Y 523.619,Z 228.204,A -85,B 0,C 180,E1 -4618.894,E2 -4618.894} C_VEL
LIN {X 0,Y 523.607,Z 225.389,A -85,B 0,C 180,E1 -4621.565,E2 -4621.565} C_VEL
LIN {X 0,Y 523.675,Z 223.257,A -85,B 0,C 180,E1 -4623.687,E2 -4623.687} C_VEL
LIN {X 0,Y 523.882,Z 223.227,A -85,B 0,C 180,E1 -4626.398,E2 -4626.398} C_VEL
LIN {X 0,Y 523.924,Z 223.224,A -85,B 0,C 180,E1 -4629.085,E2 -4629.085} C_VEL
LIN {X 0,Y 523.943,Z 223.222,A -85,B 0,C 180,E1 -4632.12,E2 -4632.12} C_VEL
LIN {X 0,Y 523.938,Z 223.22,A -85,B 0,C 180,E1 -4635.311,E2 -4635.311} C_VEL
LIN {X 0,Y 523.942,Z 223.22,A -85,B 0,C 180,E1 -4638.692,E2 -4638.692} C_VEL
LIN {X 0,Y 523.918,Z 223.223,A -85,B 0,C 180,E1 -4641.898,E2 -4641.898} C_VEL
LIN {X 0,Y 523.927,Z 223.221,A -85,B 0,C 180,E1 -4644.911,E2 -4644.911} C_VEL
LIN {X 0,Y 523.938,Z 223.225,A -85,B 0,C 180,E1 -4647.68,E2 -4647.68} C_VEL
LIN {X 0,Y 523.938,Z 223.22,A -85,B 0,C 180,E1 -4650.68,E2 -4650.68} C_VEL
LIN {X 0,Y 523.94,Z 223.219,A -85,B 0,C 180,E1 -4653.727,E2 -4653.727} C_VEL
LIN {X 0,Y 523.917,Z 223.226,A -85,B 0,C 180,E1 -4656.27,E2 -4656.27} C_VEL
LIN {X 0,Y 523.949,Z 223.218,A -85,B 0,C 180,E1 -4658.767,E2 -4658.767} C_VEL
LIN {X 0,Y 523.939,Z 223.223,A -85,B 0,C 180,E1 -4661.22,E2 -4661.22} C_VEL
LIN {X 0,Y 523.893,Z 223.225,A -85,B 0,C 180,E1 -4663.637,E2 -4663.637} C_VEL
LIN {X 0,Y 523.918,Z 223.223,A -85,B 0,C 180,E1 -4666.027,E2 -4666.027} C_VEL
LIN {X 0,Y 524.017,Z 223.215,A -85,B 0,C 180,E1 -4668.394,E2 -4668.394} C_VEL
LIN {X 0,Y 524.003,Z 223.216,A -85,B 0,C 180,E1 -4671.516,E2 -4671.516} C_VEL
LIN {X 0,Y 524.078,Z 223.203,A -85,B 0,C 180,E1 -4674.614,E2 -4674.614} C_VEL
LIN {X 0,Y 524.101,Z 223.197,A -85,B 0,C 180,E1 -4677.694,E2 -4677.694} C_VEL
LIN {X 0,Y 524.123,Z 223.197,A -85,B 0,C 180,E1 -4680.768,E2 -4680.768} C_VEL
LIN {X 0,Y 524.073,Z 223.204,A -85,B 0,C 180,E1 -4683.075,E2 -4683.075} C_VEL
LIN {X 0,Y 524.041,Z 223.207,A -85,B 0,C 180,E1 -4686.159,E2 -4686.159} C_VEL
LIN {X 0,Y 523.981,Z 223.214,A -85,B 0,C 180,E1 -4689.262,E2 -4689.262} C_VEL
LIN {X 0,Y 523.948,Z 223.221,A -85,B 0,C 180,E1 -4692.393,E2 -4692.393} C_VEL
LIN {X 0,Y 523.941,Z 223.223,A -85,B 0,C 180,E1 -4695.562,E2 -4695.562} C_VEL
LIN {X 0,Y 523.967,Z 223.216,A -85,B 0,C 180,E1 -4697.969,E2 -4697.969} C_VEL
LIN {X 0,Y 523.975,Z 223.219,A -85,B 0,C 180,E1 -4700.41,E2 -4700.41} C_VEL
LIN {X 0,Y 523.912,Z 223.223,A -85,B 0,C 180,E1 -4702.894,E2 -4702.894} C_VEL
LIN {X 0,Y 523.899,Z 223.225,A -85,B 0,C 180,E1 -4705.422,E2 -4705.422} C_VEL
LIN {X 0,Y 523.91,Z 223.224,A -85,B 0,C 180,E1 -4708.002,E2 -4708.002} C_VEL
LIN {X 0,Y 523.939,Z 223.223,A -85,B 0,C 180,E1 -4710.853,E2 -4710.853} C_VEL
LIN {X 0,Y 523.962,Z 223.218,A -85,B 0,C 180,E1 -4713.734,E2 -4713.734} C_VEL
LIN {X 0,Y 523.901,Z 223.226,A -85,B 0,C 180,E1 -4716.401,E2 -4716.401} C_VEL
LIN {X 0,Y 523.911,Z 223.224,A -85,B 0,C 180,E1 -4719.086,E2 -4719.086} C_VEL
LIN {X 0,Y 523.913,Z 223.222,A -85,B 0,C 180,E1 -4722.123,E2 -4722.123} C_VEL
LIN {X 0,Y 523.944,Z 223.219,A -85,B 0,C 180,E1 -4725.31,E2 -4725.31} C_VEL
LIN {X 0,Y 523.958,Z 223.219,A -85,B 0,C 180,E1 -4728.69,E2 -4728.69} C_VEL
LIN {X 0,Y 523.932,Z 223.323,A -85,B 0,C 180,E1 -4731.655,E2 -4731.655} C_VEL
LIN {X 0,Y 524.977,Z 229.368,A -85,B 0,C 180,E1 -4733.911,E2 -4733.911} C_VEL
LIN {X 0,Y 525.019,Z 235.585,A -85,B 0,C 180,E1 -4736.093,E2 -4736.093} C_VEL
LIN {X 0,Y 524.773,Z 244.33,A -85,B 0,C 180,E1 -4738.995,E2 -4738.995} C_VEL
LIN {X 0,Y 524.558,Z 254.075,A -85,B 0,C 180,E1 -4742.162,E2 -4742.162} C_VEL
LIN {X 0,Y 524.317,Z 262.957,A -85,B 0,C 180,E1 -4745.025,E2 -4745.025} C_VEL
LIN {X 0,Y 524.126,Z 272.225,A -85,B 0,C 180,E1 -4747.948,E2 -4747.948} C_VEL
LIN {X 0,Y 523.925,Z 281.492,A -85,B 0,C 180,E1 -4750.813,E2 -4750.813} C_VEL
LIN {X 0,Y 523.76,Z 290.759,A -85,B 0,C 180,E1 -4753.633,E2 -4753.633} C_VEL
LIN {X 0,Y 523.638,Z 299.732,A -85,B 0,C 180,E1 -4756.286,E2 -4756.286} C_VEL
LIN {X 0,Y 525.441,Z 311.268,A -85,B 0,C 180,E1 -4756.586,E2 -4756.586} C_VEL
LIN {X 0,Y 525.206,Z 323.771,A -85,B 0,C 180,E1 -4756.999,E2 -4756.999} C_VEL
LIN {X 0,Y 524.933,Z 335.411,A -85,B 0,C 180,E1 -4757.532,E2 -4757.532} C_VEL
LIN {X 0,Y 524.649,Z 346.978,A -85,B 0,C 180,E1 -4758.228,E2 -4758.228} C_VEL
LIN {X 0,Y 524.38,Z 358.262,A -85,B 0,C 180,E1 -4759.088,E2 -4759.088} C_VEL
LIN {X 0,Y 524.104,Z 367.539,A -85,B 0,C 180,E1 -4759.961,E2 -4759.961} C_VEL
LIN {X 0,Y 523.896,Z 375.991,A -85,B 0,C 180,E1 -4760.931,E2 -4760.931} C_VEL
LIN {X 0,Y 523.688,Z 384.237,A -85,B 0,C 180,E1 -4762.094,E2 -4762.094} C_VEL
LIN {X 0,Y 523.574,Z 389.869,A -85,B 0,C 180,E1 -4763.061,E2 -4763.061} C_VEL
LIN {X 0,Y 523.544,Z 395.366,A -85,B 0,C 180,E1 -4764.222,E2 -4764.222} C_VEL
LIN {X 0,Y 523.361,Z 399.677,A -85,B 0,C 180,E1 -4765.379,E2 -4765.379} C_VEL
LIN {X 0,Y 523.443,Z 401.958,A -85,B 0,C 180,E1 -4766.151,E2 -4766.151} C_VEL
LIN {X 0,Y 523.367,Z 403.808,A -85,B 0,C 180,E1 -4766.921,E2 -4766.921} C_VEL
LIN {X 0,Y 523.335,Z 405.197,A -85,B 0,C 180,E1 -4767.691,E2 -4767.691} C_VEL
LIN {X 0,Y 523.25,Z 406.785,A -85,B 0,C 180,E1 -4769.231,E2 -4769.231} C_VEL
LIN {X 0,Y 523.246,Z 407,A -85,B 0,C 180,E1 -4770,E2 -4770} C_VEL
LIN {X 0,Y 523.275,Z 406.186,A -85,B 0,C 180,E1 -4771.539,E2 -4771.539} C_VEL
LIN {X 0,Y 523.335,Z 405.198,A -85,B 0,C 180,E1 -4772.309,E2 -4772.309} C_VEL
LIN {X 0,Y 523.367,Z 403.81,A -85,B 0,C 180,E1 -4773.079,E2 -4773.079} C_VEL
LIN {X 0,Y 523.441,Z 400.895,A -85,B 0,C 180,E1 -4774.235,E2 -4774.235} C_VEL
LIN {X 0,Y 523.464,Z 396.948,A -85,B 0,C 180,E1 -4775.393,E2 -4775.393} C_VEL
LIN {X 0,Y 523.524,Z 391.722,A -85,B 0,C 180,E1 -4776.582,E2 -4776.582} C_VEL
LIN {X 0,Y 523.665,Z 385.467,A -85,B 0,C 180,E1 -4777.713,E2 -4777.713} C_VEL
LIN {X 0,Y 523.857,Z 377.477,A -85,B 0,C 180,E1 -4778.875,E2 -4778.875} C_VEL
LIN {X 0,Y 524.059,Z 369.333,A -85,B 0,C 180,E1 -4779.845,E2 -4779.845} C_VEL
LIN {X 0,Y 524.336,Z 359.398,A -85,B 0,C 180,E1 -4780.816,E2 -4780.816} C_VEL
LIN {X 0,Y 524.63,Z 348.231,A -85,B 0,C 180,E1 -4781.686,E2 -4781.686} C_VEL
LIN {X 0,Y 524.848,Z 337.172,A -85,B 0,C 180,E1 -4782.372,E2 -4782.372} C_VEL
LIN {X 0,Y 525.183,Z 324.973,A -85,B 0,C 180,E1 -4782.953,E2 -4782.953} C_VEL
LIN {X 0,Y 525.408,Z 312.168,A -85,B 0,C 180,E1 -4783.39,E2 -4783.39} C_VEL
LIN {X 0,Y 524.501,Z 304.649,A -85,B 0,C 180,E1 -4783.599,E2 -4783.599} C_VEL
LIN {X 0,Y 523.627,Z 299.529,A -85,B 0,C 180,E1 -4783.733,E2 -4783.733} C_VEL
LIN {X 0,Y 523.761,Z 290.759,A -85,B 0,C 180,E1 -4786.367,E2 -4786.367} C_VEL
LIN {X 0,Y 523.925,Z 281.491,A -85,B 0,C 180,E1 -4789.187,E2 -4789.187} C_VEL
LIN {X 0,Y 524.13,Z 271.436,A -85,B 0,C 180,E1 -4792.299,E2 -4792.299} C_VEL
LIN {X 0,Y 524.351,Z 261.633,A -85,B 0,C 180,E1 -4795.398,E2 -4795.398} C_VEL
LIN {X 0,Y 524.61,Z 252.365,A -85,B 0,C 180,E1 -4798.397,E2 -4798.397} C_VEL
LIN {X 0,Y 524.828,Z 242.869,A -85,B 0,C 180,E1 -4801.484,E2 -4801.484} C_VEL
LIN {X 0,Y 525.042,Z 234.701,A -85,B 0,C 180,E1 -4804.208,E2 -4804.208} C_VEL
LIN {X 0,Y 524.975,Z 229.322,A -85,B 0,C 180,E1 -4806.089,E2 -4806.089} C_VEL
LIN {X 0,Y 523.921,Z 223.227,A -85,B 0,C 180,E1 -4808.408,E2 -4808.408} C_VEL
LIN {X 0,Y 523.959,Z 223.219,A -85,B 0,C 180,E1 -4811.31,E2 -4811.31} C_VEL
LIN {X 0,Y 523.946,Z 223.221,A -85,B 0,C 180,E1 -4814.69,E2 -4814.69} C_VEL
LIN {X 0,Y 523.914,Z 223.222,A -85,B 0,C 180,E1 -4817.877,E2 -4817.877} C_VEL
LIN {X 0,Y 523.912,Z 223.223,A -85,B 0,C 180,E1 -4821.082,E2 -4821.082} C_VEL
LIN {X 0,Y 523.899,Z 223.227,A -85,B 0,C 180,E1 -4823.825,E2 -4823.825} C_VEL
LIN {X 0,Y 523.946,Z 223.219,A -85,B 0,C 180,E1 -4826.636,E2 -4826.636} C_VEL
LIN {X 0,Y 523.949,Z 223.221,A -85,B 0,C 180,E1 -4829.355,E2 -4829.355} C_VEL
LIN {X 0,Y 523.92,Z 223.225,A -85,B 0,C 180,E1 -4832.294,E2 -4832.294} C_VEL
LIN {X 0,Y 523.905,Z 223.224,A -85,B 0,C 180,E1 -4835.427,E2 -4835.427} C_VEL
LIN {X 0,Y 523.943,Z 223.222,A -85,B 0,C 180,E1 -4837.94,E2 -4837.94} C_VEL
LIN {X 0,Y 523.979,Z 223.215,A -85,B 0,C 180,E1 -4840.408,E2 -4840.408} C_VEL
LIN {X 0,Y 523.961,Z 223.22,A -85,B 0,C 180,E1 -4842.837,E2 -4842.837} C_VEL
LIN {X 0,Y 523.973,Z 223.215,A -85,B 0,C 180,E1 -4845.236,E2 -4845.236} C_VEL
LIN {X 0,Y 523.967,Z 223.216,A -85,B 0,C 180,E1 -4848.393,E2 -4848.393} C_VEL
LIN {X 0,Y 523.986,Z 223.218,A -85,B 0,C 180,E1 -4851.516,E2 -4851.516} C_VEL
LIN {X 0,Y 524.042,Z 223.207,A -85,B 0,C 180,E1 -4853.841,E2 -4853.841} C_VEL
LIN {X 0,Y 524.074,Z 223.204,A -85,B 0,C 180,E1 -4856.925,E2 -4856.925} C_VEL
LIN {X 0,Y 524.1,Z 223.202,A -85,B 0,C 180,E1 -4860,E2 -4860} C_VEL
LIN {X 0,Y 524.036,Z 223.21,A -85,B 0,C 180,E1 -4863.075,E2 -4863.075} C_VEL
LIN {X 0,Y 524.038,Z 223.208,A -85,B 0,C 180,E1 -4866.159,E2 -4866.159} C_VEL
LIN {X 0,Y 523.992,Z 223.213,A -85,B 0,C 180,E1 -4869.262,E2 -4869.262} C_VEL
LIN {X 0,Y 524.005,Z 223.215,A -85,B 0,C 180,E1 -4871.737,E2 -4871.737} C_VEL
LIN {X 0,Y 523.988,Z 223.217,A -85,B 0,C 180,E1 -4875.048,E2 -4875.048} C_VEL
LIN {X 0,Y 523.92,Z 223.22,A -85,B 0,C 180,E1 -4877.971,E2 -4877.971} C_VEL
LIN {X 0,Y 523.977,Z 223.219,A -85,B 0,C 180,E1 -4880.41,E2 -4880.41} C_VEL
LIN {X 0,Y 523.916,Z 223.223,A -85,B 0,C 180,E1 -4882.893,E2 -4882.893} C_VEL
LIN {X 0,Y 523.987,Z 223.215,A -85,B 0,C 180,E1 -4886.019,E2 -4886.019} C_VEL
LIN {X 0,Y 523.935,Z 223.221,A -85,B 0,C 180,E1 -4889.319,E2 -4889.319} C_VEL
LIN {X 0,Y 523.938,Z 223.224,A -85,B 0,C 180,E1 -4892.449,E2 -4892.449} C_VEL
